LIN {X 0,Y 573.221,Z 379.814,A -85,B 0,C 180,E1 -2075.627,E2 -2075.627} C_VEL
LIN {X 0,Y 573.157,Z 385.848,A -85,B 0,C 180,E1 -2078.46,E2 -2078.46} C_VEL
LIN {X 0,Y 573.104,Z 392.081,A -85,B 0,C 180,E1 -2081.313,E2 -2081.313} C_VEL
LIN {X 0,Y 573.094,Z 398.89,A -85,B 0,C 180,E1 -2084.352,E2 -2084.352} C_VEL
LIN {X 0,Y 573.007,Z 405.201,A -85,B 0,C 180,E1 -2087.117,E2 -2087.117} C_VEL
LIN {X 0,Y 572.989,Z 410.326,A -85,B 0,C 180,E1 -2089.338,E2 -2089.338} C_VEL
LIN {X 0,Y 572.956,Z 415.575,A -85,B 0,C 180,E1 -2091.589,E2 -2091.589} C_VEL
LIN {X 0,Y 572.996,Z 419.359,A -85,B 0,C 180,E1 -2093.203,E2 -2093.203} C_VEL
LIN {X 0,Y 573.514,Z 425.872,A -85,B 0,C 180,E1 -2093.384,E2 -2093.384} C_VEL
LIN {X 0,Y 573.391,Z 435.633,A -85,B 0,C 180,E1 -2093.712,E2 -2093.712} C_VEL
LIN {X 0,Y 573.301,Z 447.019,A -85,B 0,C 180,E1 -2094.245,E2 -2094.245} C_VEL
LIN {X 0,Y 573.212,Z 457.823,A -85,B 0,C 180,E1 -2094.94,E2 -2094.94} C_VEL
LIN {X 0,Y 573.204,Z 465.961,A -85,B 0,C 180,E1 -2095.605,E2 -2095.605} C_VEL
LIN {X 0,Y 573.121,Z 474.398,A -85,B 0,C 180,E1 -2096.47,E2 -2096.47} C_VEL
LIN {X 0,Y 573.107,Z 481.387,A -85,B 0,C 180,E1 -2097.376,E2 -2097.376} C_VEL
LIN {X 0,Y 573.042,Z 486.731,A -85,B 0,C 180,E1 -2098.251,E2 -2098.251} C_VEL
LIN {X 0,Y 572.997,Z 492.29,A -85,B 0,C 180,E1 -2099.444,E2 -2099.444} C_VEL
LIN {X 0,Y 572.972,Z 494.817,A -85,B 0,C 180,E1 -2100.189,E2 -2100.189} C_VEL
LIN {X 0,Y 572.968,Z 496.858,A -85,B 0,C 180,E1 -2101.006,E2 -2101.006} C_VEL
LIN {X 0,Y 572.948,Z 498.62,A -85,B 0,C 180,E1 -2102.18,E2 -2102.18} C_VEL
LIN {X 0,Y 572.953,Z 498.823,A -85,B 0,C 180,E1 -2103.5,E2 -2103.5} C_VEL
LIN {X 0,Y 572.955,Z 497.535,A -85,B 0,C 180,E1 -2104.731,E2 -2104.731} C_VEL
LIN {X 0,Y 572.995,Z 494.283,A -85,B 0,C 180,E1 -2106.065,E2 -2106.065} C_VEL
LIN {X 0,Y 573.008,Z 490.226,A -85,B 0,C 180,E1 -2107.134,E2 -2107.134} C_VEL
LIN {X 0,Y 573.067,Z 484.148,A -85,B 0,C 180,E1 -2108.29,E2 -2108.29} C_VEL
LIN {X 0,Y 573.107,Z 477.566,A -85,B 0,C 180,E1 -2109.237,E2 -2109.237} C_VEL
LIN {X 0,Y 573.156,Z 469.185,A -85,B 0,C 180,E1 -2110.182,E2 -2110.182} C_VEL
LIN {X 0,Y 573.23,Z 459.968,A -85,B 0,C 180,E1 -2110.987,E2 -2110.987} C_VEL
LIN {X 0,Y 573.289,Z 451.126,A -85,B 0,C 180,E1 -2111.6,E2 -2111.6} C_VEL
LIN {X 0,Y 573.399,Z 441.637,A -85,B 0,C 180,E1 -2112.115,E2 -2112.115} C_VEL
LIN {X 0,Y 573.462,Z 430.782,A -85,B 0,C 180,E1 -2112.559,E2 -2112.559} C_VEL
LIN {X 0,Y 573.262,Z 421.712,A -85,B 0,C 180,E1 -2112.823,E2 -2112.823} C_VEL
LIN {X 0,Y 572.984,Z 419.34,A -85,B 0,C 180,E1 -2112.895,E2 -2112.895} C_VEL
LIN {X 0,Y 573.006,Z 412.902,A -85,B 0,C 180,E1 -2115.644,E2 -2115.644} C_VEL
LIN {X 0,Y 572.99,Z 406.238,A -85,B 0,C 180,E1 -2118.522,E2 -2118.522} C_VEL
LIN {X 0,Y 573.032,Z 398.959,A -85,B 0,C 180,E1 -2121.71,E2 -2121.71} C_VEL
LIN {X 0,Y 573.049,Z 393.732,A -85,B 0,C 180,E1 -2124.037,E2 -2124.037} C_VEL
LIN {X 0,Y 573.082,Z 388.318,A -85,B 0,C 180,E1 -2126.506,E2 -2126.506} C_VEL
LIN {X 0,Y 573.121,Z 382.746,A -85,B 0,C 180,E1 -2129.131,E2 -2129.131} C_VEL
LIN {X 0,Y 573.217,Z 376.758,A -85,B 0,C 180,E1 -2131.972,E2 -2131.972} C_VEL
LIN {X 0,Y 573.242,Z 371.144,A -85,B 0,C 180,E1 -2134.59,E2 -2134.59} C_VEL
LIN {X 0,Y 573.271,Z 369.078,A -85,B 0,C 180,E1 -2135.656,E2 -2135.656} C_VEL
LIN {X 0,Y 573.247,Z 369.082,A -85,B 0,C 180,E1 -2137.663,E2 -2137.663} C_VEL
LIN {X 0,Y 573.255,Z 369.082,A -85,B 0,C 180,E1 -2140.727,E2 -2140.727} C_VEL
LIN {X 0,Y 573.237,Z 369.082,A -85,B 0,C 180,E1 -2143.622,E2 -2143.622} C_VEL
LIN {X 0,Y 573.268,Z 369.08,A -85,B 0,C 180,E1 -2145.807,E2 -2145.807} C_VEL
LIN {X 0,Y 573.31,Z 369.075,A -85,B 0,C 180,E1 -2148.707,E2 -2148.707} C_VEL
LIN {X 0,Y 573.286,Z 369.076,A -85,B 0,C 180,E1 -2151.541,E2 -2151.541} C_VEL
LIN {X 0,Y 573.287,Z 369.075,A -85,B 0,C 180,E1 -2154.372,E2 -2154.372} C_VEL
LIN {X 0,Y 573.302,Z 369.076,A -85,B 0,C 180,E1 -2157.893,E2 -2157.893} C_VEL
LIN {X 0,Y 573.324,Z 369.073,A -85,B 0,C 180,E1 -2160.703,E2 -2160.703} C_VEL
LIN {X 0,Y 573.23,Z 369.083,A -85,B 0,C 180,E1 -2163.515,E2 -2163.515} C_VEL
LIN {X 0,Y 573.289,Z 369.075,A -85,B 0,C 180,E1 -2165.628,E2 -2165.628} C_VEL
LIN {X 0,Y 573.287,Z 369.076,A -85,B 0,C 180,E1 -2168.46,E2 -2168.46} C_VEL
LIN {X 0,Y 573.301,Z 369.077,A -85,B 0,C 180,E1 -2171.312,E2 -2171.312} C_VEL
LIN {X 0,Y 573.273,Z 369.076,A -85,B 0,C 180,E1 -2174.432,E2 -2174.432} C_VEL
LIN {X 0,Y 573.279,Z 369.075,A -85,B 0,C 180,E1 -2177.111,E2 -2177.111} C_VEL
LIN {X 0,Y 573.24,Z 369.08,A -85,B 0,C 180,E1 -2180.077,E2 -2180.077} C_VEL
LIN {X 0,Y 573.249,Z 369.081,A -85,B 0,C 180,E1 -2183.155,E2 -2183.155} C_VEL
LIN {X 0,Y 573.27,Z 369.078,A -85,B 0,C 180,E1 -2186.19,E2 -2186.19} C_VEL
LIN {X 0,Y 573.223,Z 369.085,A -85,B 0,C 180,E1 -2188.566,E2 -2188.566} C_VEL
LIN {X 0,Y 573.225,Z 369.082,A -85,B 0,C 180,E1 -2190.994,E2 -2190.994} C_VEL
LIN {X 0,Y 573.269,Z 369.076,A -85,B 0,C 180,E1 -2193.53,E2 -2193.53} C_VEL
LIN {X 0,Y 573.243,Z 369.079,A -85,B 0,C 180,E1 -2196.05,E2 -2196.05} C_VEL
LIN {X 0,Y 573.236,Z 369.08,A -85,B 0,C 180,E1 -2198.702,E2 -2198.702} C_VEL
LIN {X 0,Y 573.238,Z 369.081,A -85,B 0,C 180,E1 -2201.598,E2 -2201.598} C_VEL
LIN {X 0,Y 573.224,Z 369.083,A -85,B 0,C 180,E1 -2204.335,E2 -2204.335} C_VEL
LIN {X 0,Y 573.231,Z 369.085,A -85,B 0,C 180,E1 -2207.36,E2 -2207.36} C_VEL
LIN {X 0,Y 573.237,Z 369.082,A -85,B 0,C 180,E1 -2210.395,E2 -2210.395} C_VEL
LIN {X 0,Y 573.246,Z 369.081,A -85,B 0,C 180,E1 -2213.08,E2 -2213.08} C_VEL
LIN {X 0,Y 573.267,Z 369.079,A -85,B 0,C 180,E1 -2215.674,E2 -2215.674} C_VEL
LIN {X 0,Y 573.24,Z 369.084,A -85,B 0,C 180,E1 -2218.187,E2 -2218.187} C_VEL
LIN {X 0,Y 573.243,Z 369.126,A -85,B 0,C 180,E1 -2219.116,E2 -2219.116} C_VEL
LIN {X 0,Y 573.904,Z 373.266,A -85,B 0,C 180,E1 -2220.177,E2 -2220.177} C_VEL
LIN {X 0,Y 573.767,Z 383.575,A -85,B 0,C 180,E1 -2222.658,E2 -2222.658} C_VEL
LIN {X 0,Y 573.64,Z 393.801,A -85,B 0,C 180,E1 -2225.043,E2 -2225.043} C_VEL
LIN {X 0,Y 573.492,Z 407.081,A -85,B 0,C 180,E1 -2228.054,E2 -2228.054} C_VEL
LIN {X 0,Y 573.386,Z 420.619,A -85,B 0,C 180,E1 -2231.066,E2 -2231.066} C_VEL
LIN {X 0,Y 573.26,Z 433.998,A -85,B 0,C 180,E1 -2233.99,E2 -2233.99} C_VEL
LIN {X 0,Y 573.184,Z 445.774,A -85,B 0,C 180,E1 -2236.53,E2 -2236.53} C_VEL
LIN {X 0,Y 573.138,Z 450.085,A -85,B 0,C 180,E1 -2237.453,E2 -2237.453} C_VEL
LIN {X 0,Y 573.866,Z 456.184,A -85,B 0,C 180,E1 -2237.581,E2 -2237.581} C_VEL
LIN {X 0,Y 573.81,Z 469.797,A -85,B 0,C 180,E1 -2237.917,E2 -2237.917} C_VEL
LIN {X 0,Y 573.663,Z 481.536,A -85,B 0,C 180,E1 -2238.34,E2 -2238.34} C_VEL
LIN {X 0,Y 573.553,Z 492.943,A -85,B 0,C 180,E1 -2238.89,E2 -2238.89} C_VEL
LIN {X 0,Y 573.427,Z 504.229,A -85,B 0,C 180,E1 -2239.587,E2 -2239.587} C_VEL
LIN {X 0,Y 573.333,Z 514.621,A -85,B 0,C 180,E1 -2240.387,E2 -2240.387} C_VEL
LIN {X 0,Y 573.24,Z 523.131,A -85,B 0,C 180,E1 -2241.186,E2 -2241.186} C_VEL
LIN {X 0,Y 573.159,Z 530.975,A -85,B 0,C 180,E1 -2242.073,E2 -2242.073} C_VEL
LIN {X 0,Y 573.068,Z 538.985,A -85,B 0,C 180,E1 -2243.19,E2 -2243.19} C_VEL
LIN {X 0,Y 573.07,Z 545.688,A -85,B 0,C 180,E1 -2244.371,E2 -2244.371} C_VEL
LIN {X 0,Y 573.028,Z 550.378,A -85,B 0,C 180,E1 -2245.429,E2 -2245.429} C_VEL
LIN {X 0,Y 573.022,Z 553.963,A -85,B 0,C 180,E1 -2246.486,E2 -2246.486} C_VEL
LIN {X 0,Y 572.959,Z 555.814,A -85,B 0,C 180,E1 -2247.189,E2 -2247.189} C_VEL
LIN {X 0,Y 572.939,Z 557.203,A -85,B 0,C 180,E1 -2247.893,E2 -2247.893} C_VEL
LIN {X 0,Y 572.94,Z 558.786,A -85,B 0,C 180,E1 -2249.299,E2 -2249.299} C_VEL
LIN {X 0,Y 572.938,Z 559,A -85,B 0,C 180,E1 -2250.002,E2 -2250.002} C_VEL
LIN {X 0,Y 572.946,Z 558.184,A -85,B 0,C 180,E1 -2251.407,E2 -2251.407} C_VEL
LIN {X 0,Y 572.94,Z 557.196,A -85,B 0,C 180,E1 -2252.11,E2 -2252.11} C_VEL
LIN {X 0,Y 572.959,Z 555.805,A -85,B 0,C 180,E1 -2252.814,E2 -2252.814} C_VEL
LIN {X 0,Y 573.015,Z 552.891,A -85,B 0,C 180,E1 -2253.869,E2 -2253.869} C_VEL
LIN {X 0,Y 572.963,Z 548.944,A -85,B 0,C 180,E1 -2254.927,E2 -2254.927} C_VEL
LIN {X 0,Y 573.065,Z 542.869,A -85,B 0,C 180,E1 -2256.162,E2 -2256.162} C_VEL
LIN {X 0,Y 573.121,Z 536.228,A -85,B 0,C 180,E1 -2257.222,E2 -2257.222} C_VEL
LIN {X 0,Y 573.2,Z 527.979,A -85,B 0,C 180,E1 -2258.285,E2 -2258.285} C_VEL
LIN {X 0,Y 573.288,Z 519.524,A -85,B 0,C 180,E1 -2259.172,E2 -2259.172} C_VEL
LIN {X 0,Y 573.418,Z 509.08,A -85,B 0,C 180,E1 -2260.06,E2 -2260.06} C_VEL
LIN {X 0,Y 573.518,Z 497.505,A -85,B 0,C 180,E1 -2260.849,E2 -2260.849} C_VEL
LIN {X 0,Y 573.614,Z 485.855,A -85,B 0,C 180,E1 -2261.467,E2 -2261.467} C_VEL
LIN {X 0,Y 573.742,Z 473.141,A -85,B 0,C 180,E1 -2261.976,E2 -2261.976} C_VEL
LIN {X 0,Y 573.846,Z 460.469,A -85,B 0,C 180,E1 -2262.332,E2 -2262.332} C_VEL
LIN {X 0,Y 573.702,Z 453.526,A -85,B 0,C 180,E1 -2262.47,E2 -2262.47} C_VEL
LIN {X 0,Y 573.141,Z 450.07,A -85,B 0,C 180,E1 -2262.55,E2 -2262.55} C_VEL
LIN {X 0,Y 573.219,Z 437.347,A -85,B 0,C 180,E1 -2265.285,E2 -2265.285} C_VEL
LIN {X 0,Y 573.317,Z 425.571,A -85,B 0,C 180,E1 -2267.847,E2 -2267.847} C_VEL
LIN {X 0,Y 573.428,Z 413.795,A -85,B 0,C 180,E1 -2270.446,E2 -2270.446} C_VEL
LIN {X 0,Y 573.538,Z 401.461,A -85,B 0,C 180,E1 -2273.214,E2 -2273.214} C_VEL
LIN {X 0,Y 573.677,Z 390.192,A -85,B 0,C 180,E1 -2275.78,E2 -2275.78} C_VEL
LIN {X 0,Y 573.807,Z 378.43,A -85,B 0,C 180,E1 -2278.535,E2 -2278.535} C_VEL
LIN {X 0,Y 573.776,Z 371.893,A -85,B 0,C 180,E1 -2280.146,E2 -2280.146} C_VEL
LIN {X 0,Y 573.242,Z 369.084,A -85,B 0,C 180,E1 -2280.937,E2 -2280.937} C_VEL
LIN {X 0,Y 573.27,Z 369.074,A -85,B 0,C 180,E1 -2283.524,E2 -2283.524} C_VEL
LIN {X 0,Y 573.2,Z 369.085,A -85,B 0,C 180,E1 -2286.053,E2 -2286.053} C_VEL
LIN {X 0,Y 573.241,Z 369.078,A -85,B 0,C 180,E1 -2288.703,E2 -2288.703} C_VEL
LIN {X 0,Y 573.206,Z 369.084,A -85,B 0,C 180,E1 -2291.46,E2 -2291.46} C_VEL
LIN {X 0,Y 573.208,Z 369.08,A -85,B 0,C 180,E1 -2294.337,E2 -2294.337} C_VEL
LIN {X 0,Y 573.225,Z 369.083,A -85,B 0,C 180,E1 -2297.361,E2 -2297.361} C_VEL
LIN {X 0,Y 573.241,Z 369.079,A -85,B 0,C 180,E1 -2300.392,E2 -2300.392} C_VEL
LIN {X 0,Y 573.257,Z 369.075,A -85,B 0,C 180,E1 -2303.078,E2 -2303.078} C_VEL
LIN {X 0,Y 573.266,Z 369.075,A -85,B 0,C 180,E1 -2305.671,E2 -2305.671} C_VEL
LIN {X 0,Y 573.241,Z 369.08,A -85,B 0,C 180,E1 -2308.184,E2 -2308.184} C_VEL
LIN {X 0,Y 573.242,Z 369.076,A -85,B 0,C 180,E1 -2310.633,E2 -2310.633} C_VEL
LIN {X 0,Y 573.193,Z 369.087,A -85,B 0,C 180,E1 -2313.517,E2 -2313.517} C_VEL
LIN {X 0,Y 573.198,Z 369.081,A -85,B 0,C 180,E1 -2316.133,E2 -2316.133} C_VEL
LIN {X 0,Y 573.255,Z 369.082,A -85,B 0,C 180,E1 -2318.709,E2 -2318.709} C_VEL
LIN {X 0,Y 573.223,Z 369.078,A -85,B 0,C 180,E1 -2321.411,E2 -2321.411} C_VEL
LIN {X 0,Y 573.251,Z 369.077,A -85,B 0,C 180,E1 -2323.621,E2 -2323.621} C_VEL
LIN {X 0,Y 573.274,Z 369.08,A -85,B 0,C 180,E1 -2325.807,E2 -2325.807} C_VEL
LIN {X 0,Y 573.266,Z 369.074,A -85,B 0,C 180,E1 -2328.745,E2 -2328.745} C_VEL
LIN {X 0,Y 573.231,Z 369.081,A -85,B 0,C 180,E1 -2331.539,E2 -2331.539} C_VEL
LIN {X 0,Y 573.272,Z 369.075,A -85,B 0,C 180,E1 -2334.371,E2 -2334.371} C_VEL
LIN {X 0,Y 573.12,Z 369.184,A -85,B 0,C 180,E1 -2336.792,E2 -2336.792} C_VEL
LIN {X 0,Y 573.176,Z 375.949,A -85,B 0,C 180,E1 -2339.297,E2 -2339.297} C_VEL
LIN {X 0,Y 573.181,Z 381.47,A -85,B 0,C 180,E1 -2341.405,E2 -2341.405} C_VEL
LIN {X 0,Y 573.181,Z 388.472,A -85,B 0,C 180,E1 -2344.219,E2 -2344.219} C_VEL
LIN {X 0,Y 573.166,Z 394.594,A -85,B 0,C 180,E1 -2346.685,E2 -2346.685} C_VEL
LIN {X 0,Y 573.132,Z 400.488,A -85,B 0,C 180,E1 -2349.173,E2 -2349.173} C_VEL
LIN {X 0,Y 573.085,Z 407.375,A -85,B 0,C 180,E1 -2352.033,E2 -2352.033} C_VEL
LIN {X 0,Y 573.044,Z 414.457,A -85,B 0,C 180,E1 -2354.925,E2 -2354.925} C_VEL
LIN {X 0,Y 572.995,Z 419.903,A -85,B 0,C 180,E1 -2357.119,E2 -2357.119} C_VEL
LIN {X 0,Y 572.996,Z 423.478,A -85,B 0,C 180,E1 -2358.55,E2 -2358.55} C_VEL
LIN {X 0,Y 573.845,Z 430.186,A -85,B 0,C 180,E1 -2358.706,E2 -2358.706} C_VEL
LIN {X 0,Y 573.763,Z 442.032,A -85,B 0,C 180,E1 -2359.034,E2 -2359.034} C_VEL
LIN {X 0,Y 573.627,Z 453.34,A -85,B 0,C 180,E1 -2359.468,E2 -2359.468} C_VEL
LIN {X 0,Y 573.555,Z 463.451,A -85,B 0,C 180,E1 -2359.963,E2 -2359.963} C_VEL
LIN {X 0,Y 573.438,Z 474.178,A -85,B 0,C 180,E1 -2360.631,E2 -2360.631} C_VEL
LIN {X 0,Y 573.412,Z 475.368,A -85,B 0,C 180,E1 -2360.713,E2 -2360.713} C_VEL
LIN {X 0,Y 572.656,Z 480.164,A -85,B 0,C 180,E1 -2361.052,E2 -2361.052} C_VEL
LIN {X 0,Y 569.689,Z 487.629,A -85,B 0,C 180,E1 -2361.64,E2 -2361.64} C_VEL
LIN {X 0,Y 566.796,Z 494.631,A -85,B 0,C 180,E1 -2362.291,E2 -2362.291} C_VEL
LIN {X 0,Y 566.15,Z 498.531,A -85,B 0,C 180,E1 -2362.727,E2 -2362.727} C_VEL
LIN {X 0,Y 566.032,Z 506.689,A -85,B 0,C 180,E1 -2363.799,E2 -2363.799} C_VEL
LIN {X 0,Y 565.963,Z 513.78,A -85,B 0,C 180,E1 -2364.974,E2 -2364.974} C_VEL
LIN {X 0,Y 565.925,Z 519.365,A -85,B 0,C 180,E1 -2366.159,E2 -2366.159} C_VEL
LIN {X 0,Y 565.911,Z 523.539,A -85,B 0,C 180,E1 -2367.355,E2 -2367.355} C_VEL
LIN {X 0,Y 565.879,Z 525.689,A -85,B 0,C 180,E1 -2368.16,E2 -2368.16} C_VEL
LIN {X 0,Y 565.852,Z 527.302,A -85,B 0,C 180,E1 -2368.972,E2 -2368.972} C_VEL
LIN {X 0,Y 565.87,Z 528.361,A -85,B 0,C 180,E1 -2369.788,E2 -2369.788} C_VEL
LIN {X 0,Y 565.867,Z 528.999,A -85,B 0,C 180,E1 -2371.021,E2 -2371.021} C_VEL
LIN {X 0,Y 565.848,Z 528.29,A -85,B 0,C 180,E1 -2372.372,E2 -2372.372} C_VEL
LIN {X 0,Y 565.875,Z 526.246,A -85,B 0,C 180,E1 -2373.682,E2 -2373.682} C_VEL
LIN {X 0,Y 565.884,Z 522.947,A -85,B 0,C 180,E1 -2374.946,E2 -2374.946} C_VEL
LIN {X 0,Y 565.94,Z 518.319,A -85,B 0,C 180,E1 -2376.177,E2 -2376.177} C_VEL
LIN {X 0,Y 566.013,Z 511.801,A -85,B 0,C 180,E1 -2377.475,E2 -2377.475} C_VEL
LIN {X 0,Y 566.031,Z 505.02,A -85,B 0,C 180,E1 -2378.534,E2 -2378.534} C_VEL
LIN {X 0,Y 566.13,Z 497.583,A -85,B 0,C 180,E1 -2379.48,E2 -2379.48} C_VEL
LIN {X 0,Y 566.268,Z 488.609,A -85,B 0,C 180,E1 -2380.416,E2 -2380.416} C_VEL
LIN {X 0,Y 566.369,Z 478.973,A -85,B 0,C 180,E1 -2381.24,E2 -2381.24} C_VEL
LIN {X 0,Y 566.461,Z 468.39,A -85,B 0,C 180,E1 -2381.976,E2 -2381.976} C_VEL
LIN {X 0,Y 566.598,Z 457.183,A -85,B 0,C 180,E1 -2382.593,E2 -2382.593} C_VEL
LIN {X 0,Y 566.786,Z 444.591,A -85,B 0,C 180,E1 -2383.12,E2 -2383.12} C_VEL
LIN {X 0,Y 566.924,Z 432.071,A -85,B 0,C 180,E1 -2383.492,E2 -2383.492} C_VEL
LIN {X 0,Y 566.55,Z 427.486,A -85,B 0,C 180,E1 -2383.602,E2 -2383.602} C_VEL
LIN {X 0,Y 565.911,Z 423.488,A -85,B 0,C 180,E1 -2383.695,E2 -2383.695} C_VEL
LIN {X 0,Y 565.921,Z 416.591,A -85,B 0,C 180,E1 -2386.499,E2 -2386.499} C_VEL
LIN {X 0,Y 565.949,Z 409.925,A -85,B 0,C 180,E1 -2389.244,E2 -2389.244} C_VEL
LIN {X 0,Y 565.991,Z 403.165,A -85,B 0,C 180,E1 -2392.073,E2 -2392.073} C_VEL
LIN {X 0,Y 566.075,Z 395.831,A -85,B 0,C 180,E1 -2395.172,E2 -2395.172} C_VEL
LIN {X 0,Y 566.094,Z 388.666,A -85,B 0,C 180,E1 -2398.153,E2 -2398.153} C_VEL
LIN {X 0,Y 566.089,Z 381.695,A -85,B 0,C 180,E1 -2401.04,E2 -2401.04} C_VEL
LIN {X 0,Y 566.091,Z 375.921,A -85,B 0,C 180,E1 -2403.452,E2 -2403.452} C_VEL
LIN {X 0,Y 566.204,Z 369.96,A -85,B 0,C 180,E1 -2405.916,E2 -2405.916} C_VEL
LIN {X 0,Y 566.21,Z 369.96,A -85,B 0,C 180,E1 -2408.901,E2 -2408.901} C_VEL
LIN {X 0,Y 566.189,Z 369.956,A -85,B 0,C 180,E1 -2411.171,E2 -2411.171} C_VEL
LIN {X 0,Y 566.212,Z 369.957,A -85,B 0,C 180,E1 -2413.411,E2 -2413.411} C_VEL
LIN {X 0,Y 566.198,Z 369.957,A -85,B 0,C 180,E1 -2416.358,E2 -2416.358} C_VEL
LIN {X 0,Y 566.236,Z 369.952,A -85,B 0,C 180,E1 -2418.674,E2 -2418.674} C_VEL
LIN {X 0,Y 566.227,Z 369.958,A -85,B 0,C 180,E1 -2421.433,E2 -2421.433} C_VEL
LIN {X 0,Y 566.254,Z 369.952,A -85,B 0,C 180,E1 -2424.3,E2 -2424.3} C_VEL
LIN {X 0,Y 566.28,Z 369.95,A -85,B 0,C 180,E1 -2427.865,E2 -2427.865} C_VEL
LIN {X 0,Y 566.295,Z 370.044,A -85,B 0,C 180,E1 -2430.532,E2 -2430.532} C_VEL
LIN {X 0,Y 566.195,Z 374.816,A -85,B 0,C 180,E1 -2432.844,E2 -2432.844} C_VEL
LIN {X 0,Y 566.172,Z 380.804,A -85,B 0,C 180,E1 -2435.697,E2 -2435.697} C_VEL
LIN {X 0,Y 566.083,Z 386.804,A -85,B 0,C 180,E1 -2438.566,E2 -2438.566} C_VEL
LIN {X 0,Y 566.035,Z 393.035,A -85,B 0,C 180,E1 -2441.457,E2 -2441.457} C_VEL
LIN {X 0,Y 566.019,Z 399.589,A -85,B 0,C 180,E1 -2444.422,E2 -2444.422} C_VEL
LIN {X 0,Y 565.924,Z 406.166,A -85,B 0,C 180,E1 -2447.338,E2 -2447.338} C_VEL
LIN {X 0,Y 565.91,Z 411.304,A -85,B 0,C 180,E1 -2449.589,E2 -2449.589} C_VEL
LIN {X 0,Y 565.873,Z 416.567,A -85,B 0,C 180,E1 -2451.873,E2 -2451.873} C_VEL
LIN {X 0,Y 565.912,Z 419.522,A -85,B 0,C 180,E1 -2453.087,E2 -2453.087} C_VEL
LIN {X 0,Y 566.523,Z 426.242,A -85,B 0,C 180,E1 -2453.274,E2 -2453.274} C_VEL
LIN {X 0,Y 566.391,Z 436.625,A -85,B 0,C 180,E1 -2453.635,E2 -2453.635} C_VEL
LIN {X 0,Y 566.268,Z 447.72,A -85,B 0,C 180,E1 -2454.175,E2 -2454.175} C_VEL
LIN {X 0,Y 566.176,Z 458.161,A -85,B 0,C 180,E1 -2454.863,E2 -2454.863} C_VEL
LIN {X 0,Y 566.15,Z 466.175,A -85,B 0,C 180,E1 -2455.533,E2 -2455.533} C_VEL
LIN {X 0,Y 566.05,Z 474.052,A -85,B 0,C 180,E1 -2456.348,E2 -2456.348} C_VEL
LIN {X 0,Y 566.01,Z 480.308,A -85,B 0,C 180,E1 -2457.15,E2 -2457.15} C_VEL
LIN {X 0,Y 565.949,Z 486.546,A -85,B 0,C 180,E1 -2458.154,E2 -2458.154} C_VEL
LIN {X 0,Y 565.924,Z 491.874,A -85,B 0,C 180,E1 -2459.291,E2 -2459.291} C_VEL
LIN {X 0,Y 565.891,Z 494.952,A -85,B 0,C 180,E1 -2460.195,E2 -2460.195} C_VEL
LIN {X 0,Y 565.839,Z 497.681,A -85,B 0,C 180,E1 -2461.441,E2 -2461.441} C_VEL
LIN {X 0,Y 565.841,Z 498.72,A -85,B 0,C 180,E1 -2462.372,E2 -2462.372} C_VEL
LIN {X 0,Y 565.836,Z 498.988,A -85,B 0,C 180,E1 -2463.125,E2 -2463.125} C_VEL
LIN {X 0,Y 565.855,Z 498.574,A -85,B 0,C 180,E1 -2463.977,E2 -2463.977} C_VEL
LIN {X 0,Y 565.847,Z 497.228,A -85,B 0,C 180,E1 -2464.942,E2 -2464.942} C_VEL
LIN {X 0,Y 565.917,Z 494.055,A -85,B 0,C 180,E1 -2466.175,E2 -2466.175} C_VEL
LIN {X 0,Y 565.927,Z 489.398,A -85,B 0,C 180,E1 -2467.365,E2 -2467.365} C_VEL
LIN {X 0,Y 565.984,Z 484.024,A -85,B 0,C 180,E1 -2468.376,E2 -2468.376} C_VEL
LIN {X 0,Y 566.024,Z 477.803,A -85,B 0,C 180,E1 -2469.286,E2 -2469.286} C_VEL
LIN {X 0,Y 566.099,Z 469.835,A -85,B 0,C 180,E1 -2470.205,E2 -2470.205} C_VEL
LIN {X 0,Y 566.169,Z 460.783,A -85,B 0,C 180,E1 -2471.022,E2 -2471.022} C_VEL
LIN {X 0,Y 566.269,Z 451.675,A -85,B 0,C 180,E1 -2471.671,E2 -2471.671} C_VEL
LIN {X 0,Y 566.366,Z 442.425,A -85,B 0,C 180,E1 -2472.19,E2 -2472.19} C_VEL
LIN {X 0,Y 566.459,Z 432.79,A -85,B 0,C 180,E1 -2472.603,E2 -2472.603} C_VEL
LIN {X 0,Y 566.371,Z 423.198,A -85,B 0,C 180,E1 -2472.903,E2 -2472.903} C_VEL
LIN {X 0,Y 565.917,Z 419.341,A -85,B 0,C 180,E1 -2473.019,E2 -2473.019} C_VEL
LIN {X 0,Y 565.917,Z 412.282,A -85,B 0,C 180,E1 -2476.075,E2 -2476.075} C_VEL
LIN {X 0,Y 565.902,Z 405.975,A -85,B 0,C 180,E1 -2478.837,E2 -2478.837} C_VEL
LIN {X 0,Y 565.954,Z 399.704,A -85,B 0,C 180,E1 -2481.619,E2 -2481.619} C_VEL
LIN {X 0,Y 565.962,Z 393.8,A -85,B 0,C 180,E1 -2484.294,E2 -2484.294} C_VEL
LIN {X 0,Y 566.031,Z 388.257,A -85,B 0,C 180,E1 -2486.886,E2 -2486.886} C_VEL
LIN {X 0,Y 566.061,Z 383.001,A -85,B 0,C 180,E1 -2489.4,E2 -2489.4} C_VEL
LIN {X 0,Y 566.162,Z 377.851,A -85,B 0,C 180,E1 -2491.855,E2 -2491.855} C_VEL
LIN {X 0,Y 566.204,Z 372.763,A -85,B 0,C 180,E1 -2494.251,E2 -2494.251} C_VEL
LIN {X 0,Y 566.219,Z 369.957,A -85,B 0,C 180,E1 -2495.625,E2 -2495.625} C_VEL
LIN {X 0,Y 566.192,Z 369.958,A -85,B 0,C 180,E1 -2498.576,E2 -2498.576} C_VEL
LIN {X 0,Y 566.198,Z 369.958,A -85,B 0,C 180,E1 -2501.172,E2 -2501.172} C_VEL
LIN {X 0,Y 566.189,Z 369.959,A -85,B 0,C 180,E1 -2504.153,E2 -2504.153} C_VEL
LIN {X 0,Y 566.19,Z 369.959,A -85,B 0,C 180,E1 -2506.359,E2 -2506.359} C_VEL
LIN {X 0,Y 566.256,Z 369.95,A -85,B 0,C 180,E1 -2509.271,E2 -2509.271} C_VEL
LIN {X 0,Y 566.223,Z 369.954,A -85,B 0,C 180,E1 -2512.153,E2 -2512.153} C_VEL
LIN {X 0,Y 566.272,Z 369.95,A -85,B 0,C 180,E1 -2515.016,E2 -2515.016} C_VEL
LIN {X 0,Y 566.271,Z 369.951,A -85,B 0,C 180,E1 -2517.866,E2 -2517.866} C_VEL
LIN {X 0,Y 566.292,Z 369.948,A -85,B 0,C 180,E1 -2520.711,E2 -2520.711} C_VEL
LIN {X 0,Y 566.26,Z 369.95,A -85,B 0,C 180,E1 -2522.846,E2 -2522.846} C_VEL
LIN {X 0,Y 566.256,Z 369.951,A -85,B 0,C 180,E1 -2525.699,E2 -2525.699} C_VEL
LIN {X 0,Y 566.23,Z 369.957,A -85,B 0,C 180,E1 -2528.566,E2 -2528.566} C_VEL
LIN {X 0,Y 566.24,Z 369.954,A -85,B 0,C 180,E1 -2531.455,E2 -2531.455} C_VEL
LIN {X 0,Y 566.224,Z 369.954,A -85,B 0,C 180,E1 -2534.513,E2 -2534.513} C_VEL
LIN {X 0,Y 566.235,Z 369.952,A -85,B 0,C 180,E1 -2537.331,E2 -2537.331} C_VEL
LIN {X 0,Y 566.202,Z 369.958,A -85,B 0,C 180,E1 -2540.338,E2 -2540.338} C_VEL
LIN {X 0,Y 566.208,Z 369.959,A -85,B 0,C 180,E1 -2543.403,E2 -2543.403} C_VEL
LIN {X 0,Y 566.204,Z 369.958,A -85,B 0,C 180,E1 -2545.75,E2 -2545.75} C_VEL
LIN {X 0,Y 566.187,Z 369.958,A -85,B 0,C 180,E1 -2548.205,E2 -2548.205} C_VEL
LIN {X 0,Y 566.177,Z 369.959,A -85,B 0,C 180,E1 -2550.593,E2 -2550.593} C_VEL
LIN {X 0,Y 566.21,Z 369.956,A -85,B 0,C 180,E1 -2553.103,E2 -2553.103} C_VEL
LIN {X 0,Y 566.195,Z 369.959,A -85,B 0,C 180,E1 -2555.69,E2 -2555.69} C_VEL
LIN {X 0,Y 566.202,Z 369.957,A -85,B 0,C 180,E1 -2558.561,E2 -2558.561} C_VEL
LIN {X 0,Y 566.196,Z 369.958,A -85,B 0,C 180,E1 -2561.138,E2 -2561.138} C_VEL
LIN {X 0,Y 566.186,Z 369.959,A -85,B 0,C 180,E1 -2564.037,E2 -2564.037} C_VEL
LIN {X 0,Y 566.192,Z 369.959,A -85,B 0,C 180,E1 -2567.084,E2 -2567.084} C_VEL
LIN {X 0,Y 566.215,Z 369.957,A -85,B 0,C 180,E1 -2569.805,E2 -2569.805} C_VEL
LIN {X 0,Y 566.188,Z 369.961,A -85,B 0,C 180,E1 -2572.601,E2 -2572.601} C_VEL
LIN {X 0,Y 566.213,Z 369.958,A -85,B 0,C 180,E1 -2575.185,E2 -2575.185} C_VEL
LIN {X 0,Y 566.224,Z 369.957,A -85,B 0,C 180,E1 -2577.746,E2 -2577.746} C_VEL
LIN {X 0,Y 566.227,Z 370.122,A -85,B 0,C 180,E1 -2578.918,E2 -2578.918} C_VEL
LIN {X 0,Y 566.998,Z 374.99,A -85,B 0,C 180,E1 -2580.188,E2 -2580.188} C_VEL
LIN {X 0,Y 566.775,Z 386.505,A -85,B 0,C 180,E1 -2583.011,E2 -2583.011} C_VEL
LIN {X 0,Y 566.604,Z 396.827,A -85,B 0,C 180,E1 -2585.45,E2 -2585.45} C_VEL
LIN {X 0,Y 566.501,Z 408.763,A -85,B 0,C 180,E1 -2588.152,E2 -2588.152} C_VEL
LIN {X 0,Y 566.337,Z 422.222,A -85,B 0,C 180,E1 -2591.179,E2 -2591.179} C_VEL
LIN {X 0,Y 566.229,Z 433.998,A -85,B 0,C 180,E1 -2593.786,E2 -2593.786} C_VEL
LIN {X 0,Y 566.11,Z 447.456,A -85,B 0,C 180,E1 -2596.724,E2 -2596.724} C_VEL
LIN {X 0,Y 566.083,Z 450.085,A -85,B 0,C 180,E1 -2597.294,E2 -2597.294} C_VEL
LIN {X 0,Y 566.959,Z 457.324,A -85,B 0,C 180,E1 -2597.45,E2 -2597.45} C_VEL
LIN {X 0,Y 566.863,Z 470.556,A -85,B 0,C 180,E1 -2597.789,E2 -2597.789} C_VEL
LIN {X 0,Y 566.7,Z 482.561,A -85,B 0,C 180,E1 -2598.24,E2 -2598.24} C_VEL
LIN {X 0,Y 566.548,Z 494.976,A -85,B 0,C 180,E1 -2598.868,E2 -2598.868} C_VEL
LIN {X 0,Y 566.434,Z 505.509,A -85,B 0,C 180,E1 -2599.547,E2 -2599.547} C_VEL
LIN {X 0,Y 566.3,Z 515.667,A -85,B 0,C 180,E1 -2600.357,E2 -2600.357} C_VEL
LIN {X 0,Y 566.165,Z 524.803,A -85,B 0,C 180,E1 -2601.255,E2 -2601.255} C_VEL
LIN {X 0,Y 566.079,Z 533.703,A -85,B 0,C 180,E1 -2602.332,E2 -2602.332} C_VEL
LIN {X 0,Y 565.966,Z 540.966,A -85,B 0,C 180,E1 -2603.424,E2 -2603.424} C_VEL
LIN {X 0,Y 566.003,Z 545.688,A -85,B 0,C 180,E1 -2604.301,E2 -2604.301} C_VEL
LIN {X 0,Y 565.933,Z 550.378,A -85,B 0,C 180,E1 -2605.372,E2 -2605.372} C_VEL
LIN {X 0,Y 565.926,Z 553.964,A -85,B 0,C 180,E1 -2606.442,E2 -2606.442} C_VEL
LIN {X 0,Y 565.877,Z 555.814,A -85,B 0,C 180,E1 -2607.154,E2 -2607.154} C_VEL
LIN {X 0,Y 565.846,Z 558.188,A -85,B 0,C 180,E1 -2608.578,E2 -2608.578} C_VEL
LIN {X 0,Y 565.839,Z 559,A -85,B 0,C 180,E1 -2610.002,E2 -2610.002} C_VEL
LIN {X 0,Y 565.846,Z 558.184,A -85,B 0,C 180,E1 -2611.425,E2 -2611.425} C_VEL
LIN {X 0,Y 565.878,Z 555.805,A -85,B 0,C 180,E1 -2612.849,E2 -2612.849} C_VEL
LIN {X 0,Y 565.927,Z 552.891,A -85,B 0,C 180,E1 -2613.918,E2 -2613.918} C_VEL
LIN {X 0,Y 565.878,Z 548.944,A -85,B 0,C 180,E1 -2614.989,E2 -2614.989} C_VEL
LIN {X 0,Y 566.002,Z 543.859,A -85,B 0,C 180,E1 -2616.06,E2 -2616.06} C_VEL
LIN {X 0,Y 566.042,Z 537.458,A -85,B 0,C 180,E1 -2617.134,E2 -2617.134} C_VEL
LIN {X 0,Y 566.134,Z 529.467,A -85,B 0,C 180,E1 -2618.209,E2 -2618.209} C_VEL
LIN {X 0,Y 566.23,Z 521.322,A -85,B 0,C 180,E1 -2619.107,E2 -2619.107} C_VEL
LIN {X 0,Y 566.347,Z 511.385,A -85,B 0,C 180,E1 -2620.006,E2 -2620.006} C_VEL
LIN {X 0,Y 566.518,Z 500.299,A -85,B 0,C 180,E1 -2620.807,E2 -2620.807} C_VEL
LIN {X 0,Y 566.611,Z 487.922,A -85,B 0,C 180,E1 -2621.511,E2 -2621.511} C_VEL
LIN {X 0,Y 566.78,Z 475.736,A -85,B 0,C 180,E1 -2622.034,E2 -2622.034} C_VEL
LIN {X 0,Y 566.922,Z 462.3,A -85,B 0,C 180,E1 -2622.44,E2 -2622.44} C_VEL
LIN {X 0,Y 566.751,Z 454.17,A -85,B 0,C 180,E1 -2622.616,E2 -2622.616} C_VEL
LIN {X 0,Y 566.086,Z 450.07,A -85,B 0,C 180,E1 -2622.709,E2 -2622.709} C_VEL
LIN {X 0,Y 566.177,Z 437.347,A -85,B 0,C 180,E1 -2625.48,E2 -2625.48} C_VEL
LIN {X 0,Y 566.299,Z 425.571,A -85,B 0,C 180,E1 -2628.076,E2 -2628.076} C_VEL
LIN {X 0,Y 566.416,Z 413.795,A -85,B 0,C 180,E1 -2630.71,E2 -2630.71} C_VEL
LIN {X 0,Y 566.568,Z 402.011,A -85,B 0,C 180,E1 -2633.388,E2 -2633.388} C_VEL
LIN {X 0,Y 566.702,Z 390.097,A -85,B 0,C 180,E1 -2636.121,E2 -2636.121} C_VEL
LIN {X 0,Y 566.876,Z 379.903,A -85,B 0,C 180,E1 -2638.573,E2 -2638.573} C_VEL
LIN {X 0,Y 566.873,Z 373.612,A -85,B 0,C 180,E1 -2640.14,E2 -2640.14} C_VEL
LIN {X 0,Y 566.179,Z 369.964,A -85,B 0,C 180,E1 -2641.113,E2 -2641.113} C_VEL
LIN {X 0,Y 566.219,Z 369.953,A -85,B 0,C 180,E1 -2643.735,E2 -2643.735} C_VEL
LIN {X 0,Y 566.188,Z 369.961,A -85,B 0,C 180,E1 -2646.572,E2 -2646.572} C_VEL
LIN {X 0,Y 566.217,Z 369.955,A -85,B 0,C 180,E1 -2649.686,E2 -2649.686} C_VEL
LIN {X 0,Y 566.15,Z 369.96,A -85,B 0,C 180,E1 -2652.911,E2 -2652.911} C_VEL
LIN {X 0,Y 566.158,Z 369.958,A -85,B 0,C 180,E1 -2656.054,E2 -2656.054} C_VEL
LIN {X 0,Y 566.17,Z 369.964,A -85,B 0,C 180,E1 -2658.86,E2 -2658.86} C_VEL
LIN {X 0,Y 566.212,Z 369.951,A -85,B 0,C 180,E1 -2661.443,E2 -2661.443} C_VEL
LIN {X 0,Y 566.168,Z 369.965,A -85,B 0,C 180,E1 -2664.308,E2 -2664.308} C_VEL
LIN {X 0,Y 566.208,Z 369.952,A -85,B 0,C 180,E1 -2666.897,E2 -2666.897} C_VEL
LIN {X 0,Y 566.174,Z 369.96,A -85,B 0,C 180,E1 -2669.407,E2 -2669.407} C_VEL
LIN {X 0,Y 566.174,Z 369.96,A -85,B 0,C 180,E1 -2671.855,E2 -2671.855} C_VEL
LIN {X 0,Y 566.171,Z 369.957,A -85,B 0,C 180,E1 -2674.249,E2 -2674.249} C_VEL
LIN {X 0,Y 566.175,Z 369.958,A -85,B 0,C 180,E1 -2677.368,E2 -2677.368} C_VEL
LIN {X 0,Y 566.209,Z 369.952,A -85,B 0,C 180,E1 -2679.662,E2 -2679.662} C_VEL
LIN {X 0,Y 566.203,Z 369.956,A -85,B 0,C 180,E1 -2682.668,E2 -2682.668} C_VEL
LIN {X 0,Y 566.236,Z 369.954,A -85,B 0,C 180,E1 -2685.627,E2 -2685.627} C_VEL
LIN {X 0,Y 566.237,Z 369.949,A -85,B 0,C 180,E1 -2688.676,E2 -2688.676} C_VEL
LIN {X 0,Y 566.186,Z 369.96,A -85,B 0,C 180,E1 -2691.433,E2 -2691.433} C_VEL
LIN {X 0,Y 566.239,Z 369.951,A -85,B 0,C 180,E1 -2694.301,E2 -2694.301} C_VEL
LIN {X 0,Y 566.058,Z 370.033,A -85,B 0,C 180,E1 -2696.841,E2 -2696.841} C_VEL
LIN {X 0,Y 566.146,Z 378.45,A -85,B 0,C 180,E1 -2700,E2 -2700} C_VEL
LIN {X 0,Y 566.082,Z 385.71,A -85,B 0,C 180,E1 -2702.846,E2 -2702.846} C_VEL
LIN {X 0,Y 566.144,Z 391.062,A -85,B 0,C 180,E1 -2704.985,E2 -2704.985} C_VEL
LIN {X 0,Y 566.081,Z 398.004,A -85,B 0,C 180,E1 -2707.849,E2 -2707.849} C_VEL
LIN {X 0,Y 566.032,Z 404.861,A -85,B 0,C 180,E1 -2710.733,E2 -2710.733} C_VEL
LIN {X 0,Y 565.981,Z 411.856,A -85,B 0,C 180,E1 -2713.646,E2 -2713.646} C_VEL
LIN {X 0,Y 565.93,Z 419.052,A -85,B 0,C 180,E1 -2716.596,E2 -2716.596} C_VEL
LIN {X 0,Y 565.921,Z 423.479,A -85,B 0,C 180,E1 -2718.391,E2 -2718.391} C_VEL
LIN {X 0,Y 566.918,Z 430.796,A -85,B 0,C 180,E1 -2718.569,E2 -2718.569} C_VEL
LIN {X 0,Y 566.804,Z 442.349,A -85,B 0,C 180,E1 -2718.896,E2 -2718.896} C_VEL
LIN {X 0,Y 566.657,Z 453.794,A -85,B 0,C 180,E1 -2719.345,E2 -2719.345} C_VEL
LIN {X 0,Y 566.559,Z 463.924,A -85,B 0,C 180,E1 -2719.851,E2 -2719.851} C_VEL
LIN {X 0,Y 566.436,Z 474.413,A -85,B 0,C 180,E1 -2720.518,E2 -2720.518} C_VEL
LIN {X 0,Y 566.314,Z 485.153,A -85,B 0,C 180,E1 -2721.359,E2 -2721.359} C_VEL
LIN {X 0,Y 566.209,Z 494.303,A -85,B 0,C 180,E1 -2722.245,E2 -2722.245} C_VEL
LIN {X 0,Y 566.15,Z 498.531,A -85,B 0,C 180,E1 -2722.727,E2 -2722.727} C_VEL
LIN {X 0,Y 565.486,Z 502.32,A -85,B 0,C 180,E1 -2723.182,E2 -2723.182} C_VEL
LIN {X 0,Y 562.523,Z 508.004,A -85,B 0,C 180,E1 -2723.952,E2 -2723.952} C_VEL
LIN {X 0,Y 559.544,Z 513.102,A -85,B 0,C 180,E1 -2724.774,E2 -2724.774} C_VEL
LIN {X 0,Y 558.864,Z 515.801,A -85,B 0,C 180,E1 -2725.305,E2 -2725.305} C_VEL
LIN {X 0,Y 558.846,Z 520.67,A -85,B 0,C 180,E1 -2726.434,E2 -2726.434} C_VEL
LIN {X 0,Y 558.793,Z 524.77,A -85,B 0,C 180,E1 -2727.733,E2 -2727.733} C_VEL
LIN {X 0,Y 558.753,Z 526.584,A -85,B 0,C 180,E1 -2728.552,E2 -2728.552} C_VEL
LIN {X 0,Y 558.771,Z 528.379,A -85,B 0,C 180,E1 -2729.789,E2 -2729.789} C_VEL
LIN {X 0,Y 558.764,Z 528.971,A -85,B 0,C 180,E1 -2731.208,E2 -2731.208} C_VEL
LIN {X 0,Y 558.763,Z 528.091,A -85,B 0,C 180,E1 -2732.572,E2 -2732.572} C_VEL
LIN {X 0,Y 558.781,Z 525.895,A -85,B 0,C 180,E1 -2733.89,E2 -2733.89} C_VEL
LIN {X 0,Y 558.8,Z 522.39,A -85,B 0,C 180,E1 -2735.164,E2 -2735.164} C_VEL
LIN {X 0,Y 558.855,Z 517.611,A -85,B 0,C 180,E1 -2736.404,E2 -2736.404} C_VEL
LIN {X 0,Y 558.924,Z 511.504,A -85,B 0,C 180,E1 -2737.61,E2 -2737.61} C_VEL
LIN {X 0,Y 558.993,Z 503.895,A -85,B 0,C 180,E1 -2738.784,E2 -2738.784} C_VEL
LIN {X 0,Y 559.123,Z 495.09,A -85,B 0,C 180,E1 -2739.87,E2 -2739.87} C_VEL
LIN {X 0,Y 559.263,Z 485.735,A -85,B 0,C 180,E1 -2740.803,E2 -2740.803} C_VEL
LIN {X 0,Y 559.394,Z 475.179,A -85,B 0,C 180,E1 -2741.655,E2 -2741.655} C_VEL
LIN {X 0,Y 559.529,Z 463.549,A -85,B 0,C 180,E1 -2742.403,E2 -2742.403} C_VEL
LIN {X 0,Y 559.722,Z 451.047,A -85,B 0,C 180,E1 -2743.019,E2 -2743.019} C_VEL
LIN {X 0,Y 559.915,Z 438.18,A -85,B 0,C 180,E1 -2743.483,E2 -2743.483} C_VEL
LIN {X 0,Y 559.799,Z 429.29,A -85,B 0,C 180,E1 -2743.717,E2 -2743.717} C_VEL
LIN {X 0,Y 558.819,Z 423.473,A -85,B 0,C 180,E1 -2743.865,E2 -2743.865} C_VEL
LIN {X 0,Y 558.857,Z 416.264,A -85,B 0,C 180,E1 -2746.835,E2 -2746.835} C_VEL
LIN {X 0,Y 558.904,Z 409.551,A -85,B 0,C 180,E1 -2749.639,E2 -2749.639} C_VEL
LIN {X 0,Y 558.924,Z 403.053,A -85,B 0,C 180,E1 -2752.389,E2 -2752.389} C_VEL
LIN {X 0,Y 559.017,Z 397.361,A -85,B 0,C 180,E1 -2754.804,E2 -2754.804} C_VEL
LIN {X 0,Y 559.033,Z 391.266,A -85,B 0,C 180,E1 -2757.384,E2 -2757.384} C_VEL
LIN {X 0,Y 559.008,Z 385.443,A -85,B 0,C 180,E1 -2759.808,E2 -2759.808} C_VEL
LIN {X 0,Y 559.044,Z 379.588,A -85,B 0,C 180,E1 -2762.279,E2 -2762.279} C_VEL
LIN {X 0,Y 559.102,Z 371.833,A -85,B 0,C 180,E1 -2765.491,E2 -2765.491} C_VEL
LIN {X 0,Y 559.179,Z 370.834,A -85,B 0,C 180,E1 -2765.988,E2 -2765.988} C_VEL
LIN {X 0,Y 559.175,Z 370.833,A -85,B 0,C 180,E1 -2768.623,E2 -2768.623} C_VEL
LIN {X 0,Y 559.158,Z 370.833,A -85,B 0,C 180,E1 -2770.925,E2 -2770.925} C_VEL
LIN {X 0,Y 559.165,Z 370.833,A -85,B 0,C 180,E1 -2773.947,E2 -2773.947} C_VEL
LIN {X 0,Y 559.173,Z 370.831,A -85,B 0,C 180,E1 -2776.183,E2 -2776.183} C_VEL
LIN {X 0,Y 559.193,Z 370.828,A -85,B 0,C 180,E1 -2779.132,E2 -2779.132} C_VEL
LIN {X 0,Y 559.205,Z 370.827,A -85,B 0,C 180,E1 -2782.052,E2 -2782.052} C_VEL
LIN {X 0,Y 559.241,Z 370.824,A -85,B 0,C 180,E1 -2784.952,E2 -2784.952} C_VEL
LIN {X 0,Y 559.251,Z 370.826,A -85,B 0,C 180,E1 -2787.838,E2 -2787.838} C_VEL
LIN {X 0,Y 559.268,Z 370.991,A -85,B 0,C 180,E1 -2790.538,E2 -2790.538} C_VEL
LIN {X 0,Y 559.142,Z 375.793,A -85,B 0,C 180,E1 -2792.88,E2 -2792.88} C_VEL
LIN {X 0,Y 559.125,Z 381.785,A -85,B 0,C 180,E1 -2795.769,E2 -2795.769} C_VEL
LIN {X 0,Y 559.02,Z 387.855,A -85,B 0,C 180,E1 -2798.675,E2 -2798.675} C_VEL
LIN {X 0,Y 558.998,Z 393.395,A -85,B 0,C 180,E1 -2801.29,E2 -2801.29} C_VEL
LIN {X 0,Y 558.937,Z 400.44,A -85,B 0,C 180,E1 -2804.563,E2 -2804.563} C_VEL
LIN {X 0,Y 558.838,Z 407.133,A -85,B 0,C 180,E1 -2807.565,E2 -2807.565} C_VEL
LIN {X 0,Y 558.813,Z 412.285,A -85,B 0,C 180,E1 -2809.848,E2 -2809.848} C_VEL
LIN {X 0,Y 558.784,Z 417.563,A -85,B 0,C 180,E1 -2812.165,E2 -2812.165} C_VEL
LIN {X 0,Y 558.805,Z 419.591,A -85,B 0,C 180,E1 -2812.961,E2 -2812.961} C_VEL
LIN {X 0,Y 559.544,Z 426.381,A -85,B 0,C 180,E1 -2813.155,E2 -2813.155} C_VEL
LIN {X 0,Y 559.388,Z 435.886,A -85,B 0,C 180,E1 -2813.487,E2 -2813.487} C_VEL
LIN {X 0,Y 559.262,Z 446.702,A -85,B 0,C 180,E1 -2814.004,E2 -2814.004} C_VEL
LIN {X 0,Y 559.16,Z 457.321,A -85,B 0,C 180,E1 -2814.696,E2 -2814.696} C_VEL
LIN {X 0,Y 559.102,Z 465.762,A -85,B 0,C 180,E1 -2815.399,E2 -2815.399} C_VEL
LIN {X 0,Y 558.989,Z 472.676,A -85,B 0,C 180,E1 -2816.104,E2 -2816.104} C_VEL
LIN {X 0,Y 558.939,Z 479.147,A -85,B 0,C 180,E1 -2816.912,E2 -2816.912} C_VEL
LIN {X 0,Y 558.847,Z 484.484,A -85,B 0,C 180,E1 -2817.728,E2 -2817.728} C_VEL
LIN {X 0,Y 558.833,Z 488.83,A -85,B 0,C 180,E1 -2818.545,E2 -2818.545} C_VEL
LIN {X 0,Y 558.846,Z 492.333,A -85,B 0,C 180,E1 -2819.368,E2 -2819.368} C_VEL
LIN {X 0,Y 558.808,Z 495.074,A -85,B 0,C 180,E1 -2820.201,E2 -2820.201} C_VEL
LIN {X 0,Y 558.766,Z 497.374,A -85,B 0,C 180,E1 -2821.209,E2 -2821.209} C_VEL
LIN {X 0,Y 558.744,Z 498.32,A -85,B 0,C 180,E1 -2821.887,E2 -2821.887} C_VEL
LIN {X 0,Y 558.749,Z 498.893,A -85,B 0,C 180,E1 -2822.739,E2 -2822.739} C_VEL
LIN {X 0,Y 558.76,Z 498.642,A -85,B 0,C 180,E1 -2823.888,E2 -2823.888} C_VEL
LIN {X 0,Y 558.759,Z 496.814,A -85,B 0,C 180,E1 -2825.159,E2 -2825.159} C_VEL
LIN {X 0,Y 558.846,Z 494.012,A -85,B 0,C 180,E1 -2826.23,E2 -2826.23} C_VEL
LIN {X 0,Y 558.836,Z 490.697,A -85,B 0,C 180,E1 -2827.129,E2 -2827.129} C_VEL
LIN {X 0,Y 558.887,Z 486.354,A -85,B 0,C 180,E1 -2828.034,E2 -2828.034} C_VEL
LIN {X 0,Y 558.912,Z 480.737,A -85,B 0,C 180,E1 -2828.953,E2 -2828.953} C_VEL
LIN {X 0,Y 559.02,Z 473.614,A -85,B 0,C 180,E1 -2829.876,E2 -2829.876} C_VEL
LIN {X 0,Y 559.085,Z 465.71,A -85,B 0,C 180,E1 -2830.696,E2 -2830.696} C_VEL
LIN {X 0,Y 559.19,Z 456.309,A -85,B 0,C 180,E1 -2831.469,E2 -2831.469} C_VEL
LIN {X 0,Y 559.331,Z 445.345,A -85,B 0,C 180,E1 -2832.155,E2 -2832.155} C_VEL
LIN {X 0,Y 559.436,Z 437.054,A -85,B 0,C 180,E1 -2832.556,E2 -2832.556} C_VEL
LIN {X 0,Y 559.536,Z 426.721,A -85,B 0,C 180,E1 -2832.925,E2 -2832.925} C_VEL
LIN {X 0,Y 558.809,Z 419.331,A -85,B 0,C 180,E1 -2833.152,E2 -2833.152} C_VEL
LIN {X 0,Y 558.839,Z 412.295,A -85,B 0,C 180,E1 -2836.237,E2 -2836.237} C_VEL
LIN {X 0,Y 558.852,Z 405.707,A -85,B 0,C 180,E1 -2839.161,E2 -2839.161} C_VEL
LIN {X 0,Y 558.879,Z 399.526,A -85,B 0,C 180,E1 -2841.962,E2 -2841.962} C_VEL
LIN {X 0,Y 558.922,Z 393.378,A -85,B 0,C 180,E1 -2844.813,E2 -2844.813} C_VEL
LIN {X 0,Y 558.993,Z 387.968,A -85,B 0,C 180,E1 -2847.386,E2 -2847.386} C_VEL
LIN {X 0,Y 559.048,Z 382.282,A -85,B 0,C 180,E1 -2850.155,E2 -2850.155} C_VEL
LIN {X 0,Y 559.107,Z 377.783,A -85,B 0,C 180,E1 -2852.284,E2 -2852.284} C_VEL
LIN {X 0,Y 559.19,Z 372.531,A -85,B 0,C 180,E1 -2854.804,E2 -2854.804} C_VEL
LIN {X 0,Y 559.2,Z 370.831,A -85,B 0,C 180,E1 -2855.695,E2 -2855.695} C_VEL
LIN {X 0,Y 559.155,Z 370.835,A -85,B 0,C 180,E1 -2858.623,E2 -2858.623} C_VEL
LIN {X 0,Y 559.152,Z 370.837,A -85,B 0,C 180,E1 -2860.926,E2 -2860.926} C_VEL
LIN {X 0,Y 559.151,Z 370.836,A -85,B 0,C 180,E1 -2863.948,E2 -2863.948} C_VEL
LIN {X 0,Y 559.163,Z 370.836,A -85,B 0,C 180,E1 -2866.184,E2 -2866.184} C_VEL
LIN {X 0,Y 559.235,Z 370.825,A -85,B 0,C 180,E1 -2869.135,E2 -2869.135} C_VEL
LIN {X 0,Y 559.191,Z 370.83,A -85,B 0,C 180,E1 -2872.054,E2 -2872.054} C_VEL
LIN {X 0,Y 559.245,Z 370.824,A -85,B 0,C 180,E1 -2874.953,E2 -2874.953} C_VEL
LIN {X 0,Y 559.241,Z 370.827,A -85,B 0,C 180,E1 -2877.84,E2 -2877.84} C_VEL
LIN {X 0,Y 559.261,Z 370.824,A -85,B 0,C 180,E1 -2880.72,E2 -2880.72} C_VEL
LIN {X 0,Y 559.226,Z 370.826,A -85,B 0,C 180,E1 -2882.882,E2 -2882.882} C_VEL
LIN {X 0,Y 559.225,Z 370.828,A -85,B 0,C 180,E1 -2885.77,E2 -2885.77} C_VEL
LIN {X 0,Y 559.184,Z 370.834,A -85,B 0,C 180,E1 -2888.675,E2 -2888.675} C_VEL
LIN {X 0,Y 559.191,Z 370.831,A -85,B 0,C 180,E1 -2891.601,E2 -2891.601} C_VEL
LIN {X 0,Y 559.174,Z 370.832,A -85,B 0,C 180,E1 -2894.596,E2 -2894.596} C_VEL
LIN {X 0,Y 559.189,Z 370.831,A -85,B 0,C 180,E1 -2897.556,E2 -2897.556} C_VEL
LIN {X 0,Y 559.167,Z 370.837,A -85,B 0,C 180,E1 -2900.605,E2 -2900.605} C_VEL
LIN {X 0,Y 559.145,Z 370.836,A -85,B 0,C 180,E1 -2903.717,E2 -2903.717} C_VEL
LIN {X 0,Y 559.18,Z 370.834,A -85,B 0,C 180,E1 -2906.097,E2 -2906.097} C_VEL
LIN {X 0,Y 559.146,Z 370.838,A -85,B 0,C 180,E1 -2908.531,E2 -2908.531} C_VEL
LIN {X 0,Y 559.139,Z 370.84,A -85,B 0,C 180,E1 -2911.277,E2 -2911.277} C_VEL
LIN {X 0,Y 559.161,Z 370.837,A -85,B 0,C 180,E1 -2913.953,E2 -2913.953} C_VEL
LIN {X 0,Y 559.151,Z 370.836,A -85,B 0,C 180,E1 -2916.45,E2 -2916.45} C_VEL
LIN {X 0,Y 559.163,Z 370.834,A -85,B 0,C 180,E1 -2918.935,E2 -2918.935} C_VEL
LIN {X 0,Y 559.18,Z 370.833,A -85,B 0,C 180,E1 -2921.769,E2 -2921.769} C_VEL
LIN {X 0,Y 559.125,Z 370.842,A -85,B 0,C 180,E1 -2924.741,E2 -2924.741} C_VEL
LIN {X 0,Y 559.151,Z 370.838,A -85,B 0,C 180,E1 -2927.259,E2 -2927.259} C_VEL
LIN {X 0,Y 559.174,Z 370.836,A -85,B 0,C 180,E1 -2930.137,E2 -2930.137} C_VEL
LIN {X 0,Y 559.137,Z 370.84,A -85,B 0,C 180,E1 -2932.894,E2 -2932.894} C_VEL
LIN {X 0,Y 559.154,Z 370.839,A -85,B 0,C 180,E1 -2935.559,E2 -2935.559} C_VEL
LIN {X 0,Y 559.164,Z 370.837,A -85,B 0,C 180,E1 -2938.592,E2 -2938.592} C_VEL
LIN {X 0,Y 560.048,Z 375.849,A -85,B 0,C 180,E1 -2939.983,E2 -2939.983} C_VEL
LIN {X 0,Y 559.857,Z 386.836,A -85,B 0,C 180,E1 -2942.732,E2 -2942.732} C_VEL
LIN {X 0,Y 559.582,Z 398.317,A -85,B 0,C 180,E1 -2945.517,E2 -2945.517} C_VEL
LIN {X 0,Y 559.465,Z 410.955,A -85,B 0,C 180,E1 -2948.371,E2 -2948.371} C_VEL
LIN {X 0,Y 559.307,Z 423.904,A -85,B 0,C 180,E1 -2951.314,E2 -2951.314} C_VEL
LIN {X 0,Y 559.189,Z 435.68,A -85,B 0,C 180,E1 -2953.951,E2 -2953.951} C_VEL
LIN {X 0,Y 559.078,Z 447.456,A -85,B 0,C 180,E1 -2956.554,E2 -2956.554} C_VEL
LIN {X 0,Y 559.022,Z 450.085,A -85,B 0,C 180,E1 -2957.131,E2 -2957.131} C_VEL
LIN {X 0,Y 560.039,Z 457.323,A -85,B 0,C 180,E1 -2957.293,E2 -2957.293} C_VEL
LIN {X 0,Y 559.933,Z 470.556,A -85,B 0,C 180,E1 -2957.636,E2 -2957.636} C_VEL
LIN {X 0,Y 559.755,Z 482.559,A -85,B 0,C 180,E1 -2958.092,E2 -2958.092} C_VEL
LIN {X 0,Y 559.579,Z 494.631,A -85,B 0,C 180,E1 -2958.707,E2 -2958.707} C_VEL
LIN {X 0,Y 559.426,Z 505.51,A -85,B 0,C 180,E1 -2959.415,E2 -2959.415} C_VEL
LIN {X 0,Y 559.297,Z 515.667,A -85,B 0,C 180,E1 -2960.235,E2 -2960.235} C_VEL
LIN {X 0,Y 559.133,Z 524.803,A -85,B 0,C 180,E1 -2961.144,E2 -2961.144} C_VEL
LIN {X 0,Y 559.008,Z 533.702,A -85,B 0,C 180,E1 -2962.234,E2 -2962.234} C_VEL
LIN {X 0,Y 558.923,Z 539.752,A -85,B 0,C 180,E1 -2963.142,E2 -2963.142} C_VEL
LIN {X 0,Y 558.935,Z 545.688,A -85,B 0,C 180,E1 -2964.229,E2 -2964.229} C_VEL
LIN {X 0,Y 558.826,Z 550.378,A -85,B 0,C 180,E1 -2965.313,E2 -2965.313} C_VEL
LIN {X 0,Y 558.836,Z 553.964,A -85,B 0,C 180,E1 -2966.397,E2 -2966.397} C_VEL
LIN {X 0,Y 558.799,Z 555.814,A -85,B 0,C 180,E1 -2967.118,E2 -2967.118} C_VEL
LIN {X 0,Y 558.745,Z 558.188,A -85,B 0,C 180,E1 -2968.56,E2 -2968.56} C_VEL
LIN {X 0,Y 558.74,Z 559,A -85,B 0,C 180,E1 -2970.002,E2 -2970.002} C_VEL
LIN {X 0,Y 558.745,Z 558.183,A -85,B 0,C 180,E1 -2971.443,E2 -2971.443} C_VEL
LIN {X 0,Y 558.799,Z 555.804,A -85,B 0,C 180,E1 -2972.885,E2 -2972.885} C_VEL
LIN {X 0,Y 558.844,Z 552.89,A -85,B 0,C 180,E1 -2973.968,E2 -2973.968} C_VEL
LIN {X 0,Y 558.798,Z 548.944,A -85,B 0,C 180,E1 -2975.052,E2 -2975.052} C_VEL
LIN {X 0,Y 558.922,Z 543.86,A -85,B 0,C 180,E1 -2976.137,E2 -2976.137} C_VEL
LIN {X 0,Y 558.979,Z 537.458,A -85,B 0,C 180,E1 -2977.224,E2 -2977.224} C_VEL
LIN {X 0,Y 559.098,Z 529.466,A -85,B 0,C 180,E1 -2978.313,E2 -2978.313} C_VEL
LIN {X 0,Y 559.196,Z 521.321,A -85,B 0,C 180,E1 -2979.222,E2 -2979.222} C_VEL
LIN {X 0,Y 559.348,Z 511.384,A -85,B 0,C 180,E1 -2980.133,E2 -2980.133} C_VEL
LIN {X 0,Y 559.539,Z 500.404,A -85,B 0,C 180,E1 -2980.936,E2 -2980.936} C_VEL
LIN {X 0,Y 559.639,Z 488.793,A -85,B 0,C 180,E1 -2981.611,E2 -2981.611} C_VEL
LIN {X 0,Y 559.817,Z 476.956,A -85,B 0,C 180,E1 -2982.14,E2 -2982.14} C_VEL
LIN {X 0,Y 559.994,Z 464.13,A -85,B 0,C 180,E1 -2982.55,E2 -2982.55} C_VEL
LIN {X 0,Y 559.892,Z 455.309,A -85,B 0,C 180,E1 -2982.751,E2 -2982.751} C_VEL
LIN {X 0,Y 559.025,Z 450.07,A -85,B 0,C 180,E1 -2982.872,E2 -2982.872} C_VEL
LIN {X 0,Y 559.132,Z 439.03,A -85,B 0,C 180,E1 -2985.306,E2 -2985.306} C_VEL
LIN {X 0,Y 559.274,Z 427.254,A -85,B 0,C 180,E1 -2987.932,E2 -2987.932} C_VEL
LIN {X 0,Y 559.404,Z 415.478,A -85,B 0,C 180,E1 -2990.597,E2 -2990.597} C_VEL
LIN {X 0,Y 559.552,Z 403.978,A -85,B 0,C 180,E1 -2993.224,E2 -2993.224} C_VEL
LIN {X 0,Y 559.732,Z 391.705,A -85,B 0,C 180,E1 -2996.071,E2 -2996.071} C_VEL
LIN {X 0,Y 559.979,Z 380.228,A -85,B 0,C 180,E1 -2998.895,E2 -2998.895} C_VEL
LIN {X 0,Y 559.962,Z 375.298,A -85,B 0,C 180,E1 -3000.136,E2 -3000.136} C_VEL
LIN {X 0,Y 559.171,Z 370.835,A -85,B 0,C 180,E1 -3001.367,E2 -3001.367} C_VEL
LIN {X 0,Y 559.15,Z 370.837,A -85,B 0,C 180,E1 -3004.445,E2 -3004.445} C_VEL
LIN {X 0,Y 559.14,Z 370.835,A -85,B 0,C 180,E1 -3007.639,E2 -3007.639} C_VEL
LIN {X 0,Y 559.165,Z 370.837,A -85,B 0,C 180,E1 -3009.942,E2 -3009.942} C_VEL
LIN {X 0,Y 559.098,Z 370.841,A -85,B 0,C 180,E1 -3013.191,E2 -3013.191} C_VEL
LIN {X 0,Y 559.125,Z 370.836,A -85,B 0,C 180,E1 -3015.765,E2 -3015.765} C_VEL
LIN {X 0,Y 559.13,Z 370.834,A -85,B 0,C 180,E1 -3018.226,E2 -3018.226} C_VEL
LIN {X 0,Y 559.177,Z 370.829,A -85,B 0,C 180,E1 -3021.192,E2 -3021.192} C_VEL
LIN {X 0,Y 559.144,Z 370.833,A -85,B 0,C 180,E1 -3023.789,E2 -3023.789} C_VEL
LIN {X 0,Y 559.153,Z 370.835,A -85,B 0,C 180,E1 -3026.424,E2 -3026.424} C_VEL
LIN {X 0,Y 559.154,Z 370.831,A -85,B 0,C 180,E1 -3028.98,E2 -3028.98} C_VEL
LIN {X 0,Y 559.117,Z 370.842,A -85,B 0,C 180,E1 -3031.63,E2 -3031.63} C_VEL
LIN {X 0,Y 559.117,Z 370.836,A -85,B 0,C 180,E1 -3033.899,E2 -3033.899} C_VEL
LIN {X 0,Y 559.119,Z 370.841,A -85,B 0,C 180,E1 -3037.066,E2 -3037.066} C_VEL
LIN {X 0,Y 559.178,Z 370.828,A -85,B 0,C 180,E1 -3039.395,E2 -3039.395} C_VEL
LIN {X 0,Y 559.145,Z 370.833,A -85,B 0,C 180,E1 -3041.685,E2 -3041.685} C_VEL
LIN {X 0,Y 559.168,Z 370.836,A -85,B 0,C 180,E1 -3043.948,E2 -3043.948} C_VEL
LIN {X 0,Y 559.171,Z 370.833,A -85,B 0,C 180,E1 -3046.184,E2 -3046.184} C_VEL
LIN {X 0,Y 559.184,Z 370.832,A -85,B 0,C 180,E1 -3049.133,E2 -3049.133} C_VEL
LIN {X 0,Y 559.137,Z 370.834,A -85,B 0,C 180,E1 -3052.052,E2 -3052.052} C_VEL
LIN {X 0,Y 559.24,Z 370.827,A -85,B 0,C 180,E1 -3054.953,E2 -3054.953} C_VEL
LIN {X 0,Y 558.988,Z 371.01,A -85,B 0,C 180,E1 -3056.937,E2 -3056.937} C_VEL
LIN {X 0,Y 559.099,Z 379.122,A -85,B 0,C 180,E1 -3060,E2 -3060} C_VEL
LIN {X 0,Y 559.009,Z 386.49,A -85,B 0,C 180,E1 -3062.882,E2 -3062.882} C_VEL
LIN {X 0,Y 559.089,Z 391.858,A -85,B 0,C 180,E1 -3065.048,E2 -3065.048} C_VEL
LIN {X 0,Y 559.001,Z 398.805,A -85,B 0,C 180,E1 -3067.949,E2 -3067.949} C_VEL
LIN {X 0,Y 558.969,Z 405.813,A -85,B 0,C 180,E1 -3070.871,E2 -3070.871} C_VEL
LIN {X 0,Y 558.906,Z 412.82,A -85,B 0,C 180,E1 -3073.822,E2 -3073.822} C_VEL
LIN {X 0,Y 558.85,Z 420.031,A -85,B 0,C 180,E1 -3076.812,E2 -3076.812} C_VEL
LIN {X 0,Y 558.846,Z 423.481,A -85,B 0,C 180,E1 -3078.229,E2 -3078.229} C_VEL
LIN {X 0,Y 559.99,Z 431.416,A -85,B 0,C 180,E1 -3078.427,E2 -3078.427} C_VEL
LIN {X 0,Y 559.865,Z 442.917,A -85,B 0,C 180,E1 -3078.764,E2 -3078.764} C_VEL
LIN {X 0,Y 559.691,Z 453.916,A -85,B 0,C 180,E1 -3079.204,E2 -3079.204} C_VEL
LIN {X 0,Y 559.572,Z 464.586,A -85,B 0,C 180,E1 -3079.748,E2 -3079.748} C_VEL
LIN {X 0,Y 559.404,Z 476.036,A -85,B 0,C 180,E1 -3080.5,E2 -3080.5} C_VEL
LIN {X 0,Y 559.26,Z 487.881,A -85,B 0,C 180,E1 -3081.487,E2 -3081.487} C_VEL
LIN {X 0,Y 559.113,Z 496.191,A -85,B 0,C 180,E1 -3082.348,E2 -3082.348} C_VEL
LIN {X 0,Y 559.045,Z 502.802,A -85,B 0,C 180,E1 -3083.162,E2 -3083.162} C_VEL
LIN {X 0,Y 558.943,Z 509.306,A -85,B 0,C 180,E1 -3084.12,E2 -3084.12} C_VEL
LIN {X 0,Y 558.861,Z 514.871,A -85,B 0,C 180,E1 -3085.116,E2 -3085.116} C_VEL
LIN {X 0,Y 558.864,Z 515.801,A -85,B 0,C 180,E1 -3085.305,E2 -3085.305} C_VEL
LIN {X 0,Y 558.207,Z 518.357,A -85,B 0,C 180,E1 -3085.849,E2 -3085.849} C_VEL
LIN {X 0,Y 555.316,Z 521.91,A -85,B 0,C 180,E1 -3086.754,E2 -3086.754} C_VEL
LIN {X 0,Y 552.855,Z 524.218,A -85,B 0,C 180,E1 -3087.502,E2 -3087.502} C_VEL
LIN {X 0,Y 551.784,Z 525.689,A -85,B 0,C 180,E1 -3088.09,E2 -3088.09} C_VEL
LIN {X 0,Y 551.69,Z 526.098,A -85,B 0,C 180,E1 -3088.29,E2 -3088.29} C_VEL
LIN {X 0,Y 551.66,Z 527.357,A -85,B 0,C 180,E1 -3088.954,E2 -3088.954} C_VEL
LIN {X 0,Y 551.69,Z 528.569,A -85,B 0,C 180,E1 -3089.973,E2 -3089.973} C_VEL
LIN {X 0,Y 551.653,Z 528.931,A -85,B 0,C 180,E1 -3091.397,E2 -3091.397} C_VEL
LIN {X 0,Y 551.679,Z 527.887,A -85,B 0,C 180,E1 -3092.775,E2 -3092.775} C_VEL
LIN {X 0,Y 551.694,Z 525.479,A -85,B 0,C 180,E1 -3094.102,E2 -3094.102} C_VEL
LIN {X 0,Y 551.726,Z 521.82,A -85,B 0,C 180,E1 -3095.388,E2 -3095.388} C_VEL
LIN {X 0,Y 551.808,Z 516.874,A -85,B 0,C 180,E1 -3096.64,E2 -3096.64} C_VEL
LIN {X 0,Y 551.826,Z 510.61,A -85,B 0,C 180,E1 -3097.849,E2 -3097.849} C_VEL
LIN {X 0,Y 551.962,Z 502.766,A -85,B 0,C 180,E1 -3099.04,E2 -3099.04} C_VEL
LIN {X 0,Y 552.077,Z 494.896,A -85,B 0,C 180,E1 -3100.006,E2 -3100.006} C_VEL
LIN {X 0,Y 552.246,Z 485.488,A -85,B 0,C 180,E1 -3100.95,E2 -3100.95} C_VEL
LIN {X 0,Y 552.407,Z 475.249,A -85,B 0,C 180,E1 -3101.785,E2 -3101.785} C_VEL
LIN {X 0,Y 552.572,Z 463.565,A -85,B 0,C 180,E1 -3102.548,E2 -3102.548} C_VEL
LIN {X 0,Y 552.774,Z 451.047,A -85,B 0,C 180,E1 -3103.171,E2 -3103.171} C_VEL
LIN {X 0,Y 552.959,Z 438.106,A -85,B 0,C 180,E1 -3103.645,E2 -3103.645} C_VEL
LIN {X 0,Y 552.854,Z 430.082,A -85,B 0,C 180,E1 -3103.861,E2 -3103.861} C_VEL
LIN {X 0,Y 551.75,Z 423.459,A -85,B 0,C 180,E1 -3104.037,E2 -3104.037} C_VEL
LIN {X 0,Y 551.78,Z 416.251,A -85,B 0,C 180,E1 -3107.048,E2 -3107.048} C_VEL
LIN {X 0,Y 551.819,Z 409.69,A -85,B 0,C 180,E1 -3109.832,E2 -3109.832} C_VEL
LIN {X 0,Y 551.87,Z 402.733,A -85,B 0,C 180,E1 -3112.777,E2 -3112.777} C_VEL
LIN {X 0,Y 551.931,Z 397.481,A -85,B 0,C 180,E1 -3115.039,E2 -3115.039} C_VEL
LIN {X 0,Y 551.994,Z 390.261,A -85,B 0,C 180,E1 -3118.103,E2 -3118.103} C_VEL
LIN {X 0,Y 551.979,Z 383.303,A -85,B 0,C 180,E1 -3121.063,E2 -3121.063} C_VEL
LIN {X 0,Y 551.979,Z 377.373,A -85,B 0,C 180,E1 -3123.535,E2 -3123.535} C_VEL
LIN {X 0,Y 552.115,Z 371.714,A -85,B 0,C 180,E1 -3125.961,E2 -3125.961} C_VEL
LIN {X 0,Y 552.119,Z 371.712,A -85,B 0,C 180,E1 -3129.119,E2 -3129.119} C_VEL
LIN {X 0,Y 552.086,Z 371.714,A -85,B 0,C 180,E1 -3131.442,E2 -3131.442} C_VEL
LIN {X 0,Y 552.115,Z 371.714,A -85,B 0,C 180,E1 -3133.736,E2 -3133.736} C_VEL
LIN {X 0,Y 552.137,Z 371.707,A -85,B 0,C 180,E1 -3136.003,E2 -3136.003} C_VEL
LIN {X 0,Y 552.161,Z 371.704,A -85,B 0,C 180,E1 -3138.992,E2 -3138.992} C_VEL
LIN {X 0,Y 552.159,Z 371.705,A -85,B 0,C 180,E1 -3141.95,E2 -3141.95} C_VEL
LIN {X 0,Y 552.217,Z 371.7,A -85,B 0,C 180,E1 -3144.887,E2 -3144.887} C_VEL
LIN {X 0,Y 552.222,Z 371.702,A -85,B 0,C 180,E1 -3147.81,E2 -3147.81} C_VEL
LIN {X 0,Y 552.235,Z 371.767,A -85,B 0,C 180,E1 -3150.454,E2 -3150.454} C_VEL
LIN {X 0,Y 552.089,Z 376.771,A -85,B 0,C 180,E1 -3152.917,E2 -3152.917} C_VEL
LIN {X 0,Y 552.06,Z 382.751,A -85,B 0,C 180,E1 -3155.844,E2 -3155.844} C_VEL
LIN {X 0,Y 551.969,Z 388.905,A -85,B 0,C 180,E1 -3158.787,E2 -3158.787} C_VEL
LIN {X 0,Y 551.948,Z 394.272,A -85,B 0,C 180,E1 -3161.35,E2 -3161.35} C_VEL
LIN {X 0,Y 551.853,Z 401.543,A -85,B 0,C 180,E1 -3164.754,E2 -3164.754} C_VEL
LIN {X 0,Y 551.734,Z 408.104,A -85,B 0,C 180,E1 -3167.799,E2 -3167.799} C_VEL
LIN {X 0,Y 551.7,Z 413.271,A -85,B 0,C 180,E1 -3170.115,E2 -3170.115} C_VEL
LIN {X 0,Y 551.702,Z 419.342,A -85,B 0,C 180,E1 -3172.811,E2 -3172.811} C_VEL
LIN {X 0,Y 552.528,Z 427.025,A -85,B 0,C 180,E1 -3173.047,E2 -3173.047} C_VEL
LIN {X 0,Y 552.37,Z 438.721,A -85,B 0,C 180,E1 -3173.482,E2 -3173.482} C_VEL
LIN {X 0,Y 552.222,Z 449.068,A -85,B 0,C 180,E1 -3174.03,E2 -3174.03} C_VEL
LIN {X 0,Y 552.126,Z 457.909,A -85,B 0,C 180,E1 -3174.635,E2 -3174.635} C_VEL
LIN {X 0,Y 552.054,Z 466.035,A -85,B 0,C 180,E1 -3175.328,E2 -3175.328} C_VEL
LIN {X 0,Y 551.924,Z 473.025,A -85,B 0,C 180,E1 -3176.057,E2 -3176.057} C_VEL
LIN {X 0,Y 551.871,Z 479.923,A -85,B 0,C 180,E1 -3176.946,E2 -3176.946} C_VEL
LIN {X 0,Y 551.792,Z 485.869,A -85,B 0,C 180,E1 -3177.907,E2 -3177.907} C_VEL
LIN {X 0,Y 551.734,Z 490.864,A -85,B 0,C 180,E1 -3178.947,E2 -3178.947} C_VEL
LIN {X 0,Y 551.72,Z 494.521,A -85,B 0,C 180,E1 -3179.98,E2 -3179.98} C_VEL
LIN {X 0,Y 551.691,Z 496.193,A -85,B 0,C 180,E1 -3180.632,E2 -3180.632} C_VEL
LIN {X 0,Y 551.649,Z 497.794,A -85,B 0,C 180,E1 -3181.487,E2 -3181.487} C_VEL
LIN {X 0,Y 551.667,Z 498.909,A -85,B 0,C 180,E1 -3182.774,E2 -3182.774} C_VEL
LIN {X 0,Y 551.677,Z 498.472,A -85,B 0,C 180,E1 -3184.101,E2 -3184.101} C_VEL
LIN {X 0,Y 551.657,Z 497.253,A -85,B 0,C 180,E1 -3184.977,E2 -3184.977} C_VEL
LIN {X 0,Y 551.772,Z 494.088,A -85,B 0,C 180,E1 -3186.247,E2 -3186.247} C_VEL
LIN {X 0,Y 551.76,Z 490.492,A -85,B 0,C 180,E1 -3187.228,E2 -3187.228} C_VEL
LIN {X 0,Y 551.804,Z 485.779,A -85,B 0,C 180,E1 -3188.199,E2 -3188.199} C_VEL
LIN {X 0,Y 551.835,Z 480.754,A -85,B 0,C 180,E1 -3189.025,E2 -3189.025} C_VEL
LIN {X 0,Y 551.949,Z 474.205,A -85,B 0,C 180,E1 -3189.893,E2 -3189.893} C_VEL
LIN {X 0,Y 552.028,Z 467.645,A -85,B 0,C 180,E1 -3190.605,E2 -3190.605} C_VEL
LIN {X 0,Y 552.111,Z 459.585,A -85,B 0,C 180,E1 -3191.321,E2 -3191.321} C_VEL
LIN {X 0,Y 552.243,Z 451.227,A -85,B 0,C 180,E1 -3191.919,E2 -3191.919} C_VEL
LIN {X 0,Y 552.353,Z 442.844,A -85,B 0,C 180,E1 -3192.401,E2 -3192.401} C_VEL
LIN {X 0,Y 552.464,Z 434.461,A -85,B 0,C 180,E1 -3192.78,E2 -3192.78} C_VEL
LIN {X 0,Y 552.473,Z 425.352,A -85,B 0,C 180,E1 -3193.092,E2 -3193.092} C_VEL
LIN {X 0,Y 551.733,Z 419.345,A -85,B 0,C 180,E1 -3193.276,E2 -3193.276} C_VEL
LIN {X 0,Y 551.761,Z 411.978,A -85,B 0,C 180,E1 -3196.551,E2 -3196.551} C_VEL
LIN {X 0,Y 551.757,Z 405.483,A -85,B 0,C 180,E1 -3199.488,E2 -3199.488} C_VEL
LIN {X 0,Y 551.832,Z 399.535,A -85,B 0,C 180,E1 -3202.316,E2 -3202.316} C_VEL
LIN {X 0,Y 551.855,Z 393.682,A -85,B 0,C 180,E1 -3205.035,E2 -3205.035} C_VEL
LIN {X 0,Y 551.928,Z 388.154,A -85,B 0,C 180,E1 -3207.669,E2 -3207.669} C_VEL
LIN {X 0,Y 552.017,Z 382.963,A -85,B 0,C 180,E1 -3210.23,E2 -3210.23} C_VEL
LIN {X 0,Y 552.11,Z 377.19,A -85,B 0,C 180,E1 -3213,E2 -3213} C_VEL
LIN {X 0,Y 552.177,Z 371.706,A -85,B 0,C 180,E1 -3215.716,E2 -3215.716} C_VEL
LIN {X 0,Y 552.1,Z 371.715,A -85,B 0,C 180,E1 -3218.337,E2 -3218.337} C_VEL
LIN {X 0,Y 552.135,Z 371.714,A -85,B 0,C 180,E1 -3220.674,E2 -3220.674} C_VEL
LIN {X 0,Y 552.1,Z 371.715,A -85,B 0,C 180,E1 -3223.737,E2 -3223.737} C_VEL
LIN {X 0,Y 552.126,Z 371.714,A -85,B 0,C 180,E1 -3226.004,E2 -3226.004} C_VEL
LIN {X 0,Y 552.191,Z 371.703,A -85,B 0,C 180,E1 -3228.994,E2 -3228.994} C_VEL
LIN {X 0,Y 552.143,Z 371.708,A -85,B 0,C 180,E1 -3231.952,E2 -3231.952} C_VEL
LIN {X 0,Y 552.219,Z 371.699,A -85,B 0,C 180,E1 -3234.889,E2 -3234.889} C_VEL
LIN {X 0,Y 552.211,Z 371.702,A -85,B 0,C 180,E1 -3237.812,E2 -3237.812} C_VEL
LIN {X 0,Y 552.23,Z 371.699,A -85,B 0,C 180,E1 -3240.729,E2 -3240.729} C_VEL
LIN {X 0,Y 552.192,Z 371.703,A -85,B 0,C 180,E1 -3242.918,E2 -3242.918} C_VEL
LIN {X 0,Y 552.194,Z 371.704,A -85,B 0,C 180,E1 -3245.844,E2 -3245.844} C_VEL
LIN {X 0,Y 552.153,Z 371.709,A -85,B 0,C 180,E1 -3248.786,E2 -3248.786} C_VEL
LIN {X 0,Y 552.144,Z 371.708,A -85,B 0,C 180,E1 -3251.751,E2 -3251.751} C_VEL
LIN {X 0,Y 552.114,Z 371.711,A -85,B 0,C 180,E1 -3254.749,E2 -3254.749} C_VEL
LIN {X 0,Y 552.121,Z 371.713,A -85,B 0,C 180,E1 -3257.788,E2 -3257.788} C_VEL
LIN {X 0,Y 552.114,Z 371.712,A -85,B 0,C 180,E1 -3260.102,E2 -3260.102} C_VEL
LIN {X 0,Y 552.094,Z 371.714,A -85,B 0,C 180,E1 -3262.451,E2 -3262.451} C_VEL
LIN {X 0,Y 552.135,Z 371.709,A -85,B 0,C 180,E1 -3265.352,E2 -3265.352} C_VEL
LIN {X 0,Y 552.107,Z 371.712,A -85,B 0,C 180,E1 -3268.099,E2 -3268.099} C_VEL
LIN {X 0,Y 552.096,Z 371.713,A -85,B 0,C 180,E1 -3270.61,E2 -3270.61} C_VEL
LIN {X 0,Y 552.11,Z 371.712,A -85,B 0,C 180,E1 -3273.186,E2 -3273.186} C_VEL
LIN {X 0,Y 552.096,Z 371.714,A -85,B 0,C 180,E1 -3275.843,E2 -3275.843} C_VEL
LIN {X 0,Y 552.111,Z 371.713,A -85,B 0,C 180,E1 -3279.064,E2 -3279.064} C_VEL
LIN {X 0,Y 552.126,Z 371.71,A -85,B 0,C 180,E1 -3281.446,E2 -3281.446} C_VEL
LIN {X 0,Y 552.082,Z 371.718,A -85,B 0,C 180,E1 -3284.534,E2 -3284.534} C_VEL
LIN {X 0,Y 552.117,Z 371.714,A -85,B 0,C 180,E1 -3287.586,E2 -3287.586} C_VEL
LIN {X 0,Y 552.123,Z 371.712,A -85,B 0,C 180,E1 -3290.475,E2 -3290.475} C_VEL
LIN {X 0,Y 552.104,Z 371.714,A -85,B 0,C 180,E1 -3293.318,E2 -3293.318} C_VEL
LIN {X 0,Y 552.132,Z 371.711,A -85,B 0,C 180,E1 -3295.942,E2 -3295.942} C_VEL
LIN {X 0,Y 552.161,Z 371.884,A -85,B 0,C 180,E1 -3298.45,E2 -3298.45} C_VEL
LIN {X 0,Y 553.058,Z 376.695,A -85,B 0,C 180,E1 -3299.782,E2 -3299.782} C_VEL
LIN {X 0,Y 552.954,Z 385.202,A -85,B 0,C 180,E1 -3301.951,E2 -3301.951} C_VEL
LIN {X 0,Y 552.659,Z 396.915,A -85,B 0,C 180,E1 -3304.861,E2 -3304.861} C_VEL
LIN {X 0,Y 552.499,Z 406.727,A -85,B 0,C 180,E1 -3307.174,E2 -3307.174} C_VEL
LIN {X 0,Y 552.346,Z 418.802,A -85,B 0,C 180,E1 -3309.909,E2 -3309.909} C_VEL
LIN {X 0,Y 552.213,Z 432.315,A -85,B 0,C 180,E1 -3312.981,E2 -3312.981} C_VEL
LIN {X 0,Y 552.049,Z 445.774,A -85,B 0,C 180,E1 -3316.004,E2 -3316.004} C_VEL
LIN {X 0,Y 551.978,Z 450.085,A -85,B 0,C 180,E1 -3316.964,E2 -3316.964} C_VEL
LIN {X 0,Y 553.075,Z 458.461,A -85,B 0,C 180,E1 -3317.153,E2 -3317.153} C_VEL
LIN {X 0,Y 552.988,Z 470.555,A -85,B 0,C 180,E1 -3317.478,E2 -3317.478} C_VEL
LIN {X 0,Y 552.808,Z 482.549,A -85,B 0,C 180,E1 -3317.94,E2 -3317.94} C_VEL
LIN {X 0,Y 552.621,Z 493.291,A -85,B 0,C 180,E1 -3318.484,E2 -3318.484} C_VEL
LIN {X 0,Y 552.478,Z 504.225,A -85,B 0,C 180,E1 -3319.187,E2 -3319.187} C_VEL
LIN {X 0,Y 552.303,Z 514.624,A -85,B 0,C 180,E1 -3320.018,E2 -3320.018} C_VEL
LIN {X 0,Y 552.13,Z 523.131,A -85,B 0,C 180,E1 -3320.847,E2 -3320.847} C_VEL
LIN {X 0,Y 552.012,Z 530.975,A -85,B 0,C 180,E1 -3321.767,E2 -3321.767} C_VEL
LIN {X 0,Y 551.888,Z 538.633,A -85,B 0,C 180,E1 -3322.869,E2 -3322.869} C_VEL
LIN {X 0,Y 551.867,Z 545.688,A -85,B 0,C 180,E1 -3324.154,E2 -3324.154} C_VEL
LIN {X 0,Y 551.725,Z 550.379,A -85,B 0,C 180,E1 -3325.252,E2 -3325.252} C_VEL
LIN {X 0,Y 551.75,Z 553.965,A -85,B 0,C 180,E1 -3326.35,E2 -3326.35} C_VEL
LIN {X 0,Y 551.723,Z 555.814,A -85,B 0,C 180,E1 -3327.081,E2 -3327.081} C_VEL
LIN {X 0,Y 551.645,Z 558.187,A -85,B 0,C 180,E1 -3328.542,E2 -3328.542} C_VEL
LIN {X 0,Y 551.64,Z 559,A -85,B 0,C 180,E1 -3330.002,E2 -3330.002} C_VEL
LIN {X 0,Y 551.645,Z 558.182,A -85,B 0,C 180,E1 -3331.462,E2 -3331.462} C_VEL
LIN {X 0,Y 551.724,Z 555.804,A -85,B 0,C 180,E1 -3332.922,E2 -3332.922} C_VEL
LIN {X 0,Y 551.764,Z 552.89,A -85,B 0,C 180,E1 -3334.019,E2 -3334.019} C_VEL
LIN {X 0,Y 551.724,Z 548.944,A -85,B 0,C 180,E1 -3335.117,E2 -3335.117} C_VEL
LIN {X 0,Y 551.825,Z 543.189,A -85,B 0,C 180,E1 -3336.341,E2 -3336.341} C_VEL
LIN {X 0,Y 551.928,Z 536.227,A -85,B 0,C 180,E1 -3337.501,E2 -3337.501} C_VEL
LIN {X 0,Y 552.079,Z 527.98,A -85,B 0,C 180,E1 -3338.604,E2 -3338.604} C_VEL
LIN {X 0,Y 552.202,Z 519.525,A -85,B 0,C 180,E1 -3339.525,E2 -3339.525} C_VEL
LIN {X 0,Y 552.399,Z 509.078,A -85,B 0,C 180,E1 -3340.447,E2 -3340.447} C_VEL
LIN {X 0,Y 552.596,Z 497.255,A -85,B 0,C 180,E1 -3341.281,E2 -3341.281} C_VEL
LIN {X 0,Y 552.75,Z 485.462,A -85,B 0,C 180,E1 -3341.925,E2 -3341.925} C_VEL
LIN {X 0,Y 552.935,Z 473.137,A -85,B 0,C 180,E1 -3342.433,E2 -3342.433} C_VEL
LIN {X 0,Y 553.064,Z 460.468,A -85,B 0,C 180,E1 -3342.803,E2 -3342.803} C_VEL
LIN {X 0,Y 552.935,Z 456.021,A -85,B 0,C 180,E1 -3342.9,E2 -3342.9} C_VEL
LIN {X 0,Y 551.98,Z 450.07,A -85,B 0,C 180,E1 -3343.04,E2 -3343.04} C_VEL
LIN {X 0,Y 552.134,Z 437.347,A -85,B 0,C 180,E1 -3345.884,E2 -3345.884} C_VEL
LIN {X 0,Y 552.27,Z 425.571,A -85,B 0,C 180,E1 -3348.552,E2 -3348.552} C_VEL
LIN {X 0,Y 552.474,Z 412.024,A -85,B 0,C 180,E1 -3351.649,E2 -3351.649} C_VEL
LIN {X 0,Y 552.695,Z 398.421,A -85,B 0,C 180,E1 -3354.812,E2 -3354.812} C_VEL
LIN {X 0,Y 552.976,Z 385.189,A -85,B 0,C 180,E1 -3358.051,E2 -3358.051} C_VEL
LIN {X 0,Y 553.152,Z 378.611,A -85,B 0,C 180,E1 -3359.704,E2 -3359.704} C_VEL
LIN {X 0,Y 552.202,Z 372.076,A -85,B 0,C 180,E1 -3361.455,E2 -3361.455} C_VEL
LIN {X 0,Y 552.124,Z 371.71,A -85,B 0,C 180,E1 -3361.674,E2 -3361.674} C_VEL
LIN {X 0,Y 552.14,Z 371.709,A -85,B 0,C 180,E1 -3364.171,E2 -3364.171} C_VEL
LIN {X 0,Y 552.105,Z 371.713,A -85,B 0,C 180,E1 -3366.748,E2 -3366.748} C_VEL
LIN {X 0,Y 552.133,Z 371.708,A -85,B 0,C 180,E1 -3369.528,E2 -3369.528} C_VEL
LIN {X 0,Y 552.085,Z 371.713,A -85,B 0,C 180,E1 -3372.431,E2 -3372.431} C_VEL
LIN {X 0,Y 552.076,Z 371.716,A -85,B 0,C 180,E1 -3375.56,E2 -3375.56} C_VEL
LIN {X 0,Y 552.08,Z 371.715,A -85,B 0,C 180,E1 -3378.55,E2 -3378.55} C_VEL
LIN {X 0,Y 552.12,Z 371.707,A -85,B 0,C 180,E1 -3381.411,E2 -3381.411} C_VEL
LIN {X 0,Y 552.091,Z 371.716,A -85,B 0,C 180,E1 -3384.156,E2 -3384.156} C_VEL
LIN {X 0,Y 552.112,Z 371.709,A -85,B 0,C 180,E1 -3386.814,E2 -3386.814} C_VEL
LIN {X 0,Y 552.097,Z 371.713,A -85,B 0,C 180,E1 -3389.39,E2 -3389.39} C_VEL
LIN {X 0,Y 552.063,Z 371.717,A -85,B 0,C 180,E1 -3391.899,E2 -3391.899} C_VEL
LIN {X 0,Y 552.065,Z 371.716,A -85,B 0,C 180,E1 -3394.671,E2 -3394.671} C_VEL
LIN {X 0,Y 552.091,Z 371.711,A -85,B 0,C 180,E1 -3397.549,E2 -3397.549} C_VEL
LIN {X 0,Y 552.148,Z 371.711,A -85,B 0,C 180,E1 -3400.375,E2 -3400.375} C_VEL
LIN {X 0,Y 552.159,Z 371.703,A -85,B 0,C 180,E1 -3402.977,E2 -3402.977} C_VEL
LIN {X 0,Y 552.137,Z 371.712,A -85,B 0,C 180,E1 -3406.004,E2 -3406.004} C_VEL
LIN {X 0,Y 552.156,Z 371.706,A -85,B 0,C 180,E1 -3408.993,E2 -3408.993} C_VEL
LIN {X 0,Y 552.107,Z 371.71,A -85,B 0,C 180,E1 -3411.951,E2 -3411.951} C_VEL
LIN {X 0,Y 552.215,Z 371.703,A -85,B 0,C 180,E1 -3414.889,E2 -3414.889} C_VEL
LIN {X 0,Y 551.92,Z 371.89,A -85,B 0,C 180,E1 -3416.989,E2 -3416.989} C_VEL
LIN {X 0,Y 552.052,Z 379.801,A -85,B 0,C 180,E1 -3420,E2 -3420} C_VEL
LIN {X 0,Y 551.935,Z 387.253,A -85,B 0,C 180,E1 -3422.919,E2 -3422.919} C_VEL
LIN {X 0,Y 552.014,Z 392.657,A -85,B 0,C 180,E1 -3425.113,E2 -3425.113} C_VEL
LIN {X 0,Y 551.939,Z 399.604,A -85,B 0,C 180,E1 -3428.051,E2 -3428.051} C_VEL
LIN {X 0,Y 551.91,Z 407.476,A -85,B 0,C 180,E1 -3431.328,E2 -3431.328} C_VEL
LIN {X 0,Y 551.821,Z 415.571,A -85,B 0,C 180,E1 -3434.757,E2 -3434.757} C_VEL
LIN {X 0,Y 551.726,Z 422.855,A -85,B 0,C 180,E1 -3437.801,E2 -3437.801} C_VEL
LIN {X 0,Y 551.734,Z 423.489,A -85,B 0,C 180,E1 -3438.064,E2 -3438.064} C_VEL
LIN {X 0,Y 553.047,Z 432.027,A -85,B 0,C 180,E1 -3438.284,E2 -3438.284} C_VEL
LIN {X 0,Y 552.934,Z 443.326,A -85,B 0,C 180,E1 -3438.623,E2 -3438.623} C_VEL
LIN {X 0,Y 552.73,Z 454.137,A -85,B 0,C 180,E1 -3439.063,E2 -3439.063} C_VEL
LIN {X 0,Y 552.632,Z 463.566,A -85,B 0,C 180,E1 -3439.544,E2 -3439.544} C_VEL
LIN {X 0,Y 552.446,Z 473.503,A -85,B 0,C 180,E1 -3440.186,E2 -3440.186} C_VEL
LIN {X 0,Y 552.334,Z 482.337,A -85,B 0,C 180,E1 -3440.871,E2 -3440.871} C_VEL
LIN {X 0,Y 552.178,Z 491.231,A -85,B 0,C 180,E1 -3441.7,E2 -3441.7} C_VEL
LIN {X 0,Y 552.046,Z 499.668,A -85,B 0,C 180,E1 -3442.65,E2 -3442.65} C_VEL
LIN {X 0,Y 551.915,Z 507.624,A -85,B 0,C 180,E1 -3443.754,E2 -3443.754} C_VEL
LIN {X 0,Y 551.827,Z 513.944,A -85,B 0,C 180,E1 -3444.852,E2 -3444.852} C_VEL
LIN {X 0,Y 551.756,Z 519.507,A -85,B 0,C 180,E1 -3446.068,E2 -3446.068} C_VEL
LIN {X 0,Y 551.724,Z 523.631,A -85,B 0,C 180,E1 -3447.295,E2 -3447.295} C_VEL
LIN {X 0,Y 551.69,Z 526.098,A -85,B 0,C 180,E1 -3448.29,E2 -3448.29} C_VEL
LIN {X 0,Y 550.996,Z 527.263,A -85,B 0,C 180,E1 -3448.889,E2 -3448.889} C_VEL
LIN {X 0,Y 548.096,Z 528.489,A -85,B 0,C 180,E1 -3449.87,E2 -3449.87} C_VEL
LIN {X 0,Y 545.662,Z 528.928,A -85,B 0,C 180,E1 -3450.665,E2 -3450.665} C_VEL
LIN {X 0,Y 544.625,Z 528.964,A -85,B 0,C 180,E1 -3451.28,E2 -3451.28} C_VEL
LIN {X 0,Y 544.544,Z 528.911,A -85,B 0,C 180,E1 -3451.488,E2 -3451.488} C_VEL
LIN {X 0,Y 544.578,Z 527.622,A -85,B 0,C 180,E1 -3452.98,E2 -3452.98} C_VEL
LIN {X 0,Y 544.609,Z 525.058,A -85,B 0,C 180,E1 -3454.319,E2 -3454.319} C_VEL
LIN {X 0,Y 544.635,Z 521.258,A -85,B 0,C 180,E1 -3455.613,E2 -3455.613} C_VEL
LIN {X 0,Y 544.738,Z 516.109,A -85,B 0,C 180,E1 -3456.879,E2 -3456.879} C_VEL
LIN {X 0,Y 544.786,Z 509.653,A -85,B 0,C 180,E1 -3458.1,E2 -3458.1} C_VEL
LIN {X 0,Y 544.95,Z 501.594,A -85,B 0,C 180,E1 -3459.303,E2 -3459.303} C_VEL
LIN {X 0,Y 545.096,Z 493.181,A -85,B 0,C 180,E1 -3460.31,E2 -3460.31} C_VEL
LIN {X 0,Y 545.273,Z 483.79,A -85,B 0,C 180,E1 -3461.231,E2 -3461.231} C_VEL
LIN {X 0,Y 545.454,Z 473.32,A -85,B 0,C 180,E1 -3462.067,E2 -3462.067} C_VEL
LIN {X 0,Y 545.624,Z 462.434,A -85,B 0,C 180,E1 -3462.76,E2 -3462.76} C_VEL
LIN {X 0,Y 545.839,Z 450.584,A -85,B 0,C 180,E1 -3463.348,E2 -3463.348} C_VEL
LIN {X 0,Y 546.044,Z 437.551,A -85,B 0,C 180,E1 -3463.824,E2 -3463.824} C_VEL
LIN {X 0,Y 545.925,Z 431.134,A -85,B 0,C 180,E1 -3464.001,E2 -3464.001} C_VEL
LIN {X 0,Y 544.669,Z 423.473,A -85,B 0,C 180,E1 -3464.204,E2 -3464.204} C_VEL
LIN {X 0,Y 544.698,Z 417.206,A -85,B 0,C 180,E1 -3466.855,E2 -3466.855} C_VEL
LIN {X 0,Y 544.75,Z 410.373,A -85,B 0,C 180,E1 -3469.828,E2 -3469.828} C_VEL
LIN {X 0,Y 544.788,Z 403.589,A -85,B 0,C 180,E1 -3472.675,E2 -3472.675} C_VEL
LIN {X 0,Y 544.864,Z 397.283,A -85,B 0,C 180,E1 -3475.42,E2 -3475.42} C_VEL
LIN {X 0,Y 544.941,Z 390.438,A -85,B 0,C 180,E1 -3478.341,E2 -3478.341} C_VEL
LIN {X 0,Y 544.942,Z 383.056,A -85,B 0,C 180,E1 -3481.497,E2 -3481.497} C_VEL
LIN {X 0,Y 544.963,Z 375.888,A -85,B 0,C 180,E1 -3484.52,E2 -3484.52} C_VEL
LIN {X 0,Y 545.071,Z 372.591,A -85,B 0,C 180,E1 -3485.988,E2 -3485.988} C_VEL
LIN {X 0,Y 545.066,Z 372.593,A -85,B 0,C 180,E1 -3488.835,E2 -3488.835} C_VEL
LIN {X 0,Y 545.051,Z 372.59,A -85,B 0,C 180,E1 -3491.193,E2 -3491.193} C_VEL
LIN {X 0,Y 545.066,Z 372.593,A -85,B 0,C 180,E1 -3493.52,E2 -3493.52} C_VEL
LIN {X 0,Y 545.097,Z 372.584,A -85,B 0,C 180,E1 -3495.819,E2 -3495.819} C_VEL
LIN {X 0,Y 545.118,Z 372.582,A -85,B 0,C 180,E1 -3498.848,E2 -3498.848} C_VEL
LIN {X 0,Y 545.129,Z 372.581,A -85,B 0,C 180,E1 -3501.846,E2 -3501.846} C_VEL
LIN {X 0,Y 545.194,Z 372.576,A -85,B 0,C 180,E1 -3504.821,E2 -3504.821} C_VEL
LIN {X 0,Y 545.193,Z 372.577,A -85,B 0,C 180,E1 -3507.782,E2 -3507.782} C_VEL
LIN {X 0,Y 545.208,Z 372.721,A -85,B 0,C 180,E1 -3510.46,E2 -3510.46} C_VEL
LIN {X 0,Y 545.182,Z 376.24,A -85,B 0,C 180,E1 -3512.215,E2 -3512.215} C_VEL
LIN {X 0,Y 545.018,Z 382.21,A -85,B 0,C 180,E1 -3515.177,E2 -3515.177} C_VEL
LIN {X 0,Y 544.941,Z 388.34,A -85,B 0,C 180,E1 -3518.154,E2 -3518.154} C_VEL
LIN {X 0,Y 544.881,Z 395.132,A -85,B 0,C 180,E1 -3521.403,E2 -3521.403} C_VEL
LIN {X 0,Y 544.823,Z 402.024,A -85,B 0,C 180,E1 -3524.655,E2 -3524.655} C_VEL
LIN {X 0,Y 544.711,Z 407.595,A -85,B 0,C 180,E1 -3527.3,E2 -3527.3} C_VEL
LIN {X 0,Y 544.62,Z 414.253,A -85,B 0,C 180,E1 -3530.388,E2 -3530.388} C_VEL
LIN {X 0,Y 544.609,Z 419.336,A -85,B 0,C 180,E1 -3532.674,E2 -3532.674} C_VEL
LIN {X 0,Y 545.542,Z 427.542,A -85,B 0,C 180,E1 -3532.933,E2 -3532.933} C_VEL
LIN {X 0,Y 545.37,Z 439.462,A -85,B 0,C 180,E1 -3533.393,E2 -3533.393} C_VEL
LIN {X 0,Y 545.197,Z 449.452,A -85,B 0,C 180,E1 -3533.938,E2 -3533.938} C_VEL
LIN {X 0,Y 545.081,Z 458.423,A -85,B 0,C 180,E1 -3534.568,E2 -3534.568} C_VEL
LIN {X 0,Y 545.01,Z 465.562,A -85,B 0,C 180,E1 -3535.182,E2 -3535.182} C_VEL
LIN {X 0,Y 544.854,Z 473.377,A -85,B 0,C 180,E1 -3536.01,E2 -3536.01} C_VEL
LIN {X 0,Y 544.809,Z 479.712,A -85,B 0,C 180,E1 -3536.837,E2 -3536.837} C_VEL
LIN {X 0,Y 544.692,Z 484.946,A -85,B 0,C 180,E1 -3537.675,E2 -3537.675} C_VEL
LIN {X 0,Y 544.658,Z 489.197,A -85,B 0,C 180,E1 -3538.515,E2 -3538.515} C_VEL
LIN {X 0,Y 544.673,Z 492.609,A -85,B 0,C 180,E1 -3539.359,E2 -3539.359} C_VEL
LIN {X 0,Y 544.626,Z 495.283,A -85,B 0,C 180,E1 -3540.214,E2 -3540.214} C_VEL
LIN {X 0,Y 544.56,Z 497.234,A -85,B 0,C 180,E1 -3541.077,E2 -3541.077} C_VEL
LIN {X 0,Y 544.552,Z 498.437,A -85,B 0,C 180,E1 -3541.945,E2 -3541.945} C_VEL
LIN {X 0,Y 544.564,Z 498.992,A -85,B 0,C 180,E1 -3542.979,E2 -3542.979} C_VEL
LIN {X 0,Y 544.577,Z 498.217,A -85,B 0,C 180,E1 -3544.316,E2 -3544.316} C_VEL
LIN {X 0,Y 544.587,Z 495.912,A -85,B 0,C 180,E1 -3545.608,E2 -3545.608} C_VEL
LIN {X 0,Y 544.663,Z 493.691,A -85,B 0,C 180,E1 -3546.407,E2 -3546.407} C_VEL
LIN {X 0,Y 544.697,Z 490.282,A -85,B 0,C 180,E1 -3547.328,E2 -3547.328} C_VEL
LIN {X 0,Y 544.741,Z 485.806,A -85,B 0,C 180,E1 -3548.26,E2 -3548.26} C_VEL
LIN {X 0,Y 544.775,Z 481.679,A -85,B 0,C 180,E1 -3548.967,E2 -3548.967} C_VEL
LIN {X 0,Y 544.886,Z 474.701,A -85,B 0,C 180,E1 -3549.921,E2 -3549.921} C_VEL
LIN {X 0,Y 544.961,Z 468.084,A -85,B 0,C 180,E1 -3550.659,E2 -3550.659} C_VEL
LIN {X 0,Y 545.071,Z 460.435,A -85,B 0,C 180,E1 -3551.358,E2 -3551.358} C_VEL
LIN {X 0,Y 545.201,Z 452.715,A -85,B 0,C 180,E1 -3551.936,E2 -3551.936} C_VEL
LIN {X 0,Y 545.329,Z 444.354,A -85,B 0,C 180,E1 -3552.442,E2 -3552.442} C_VEL
LIN {X 0,Y 545.445,Z 435.407,A -85,B 0,C 180,E1 -3552.868,E2 -3552.868} C_VEL
LIN {X 0,Y 545.495,Z 426.045,A -85,B 0,C 180,E1 -3553.201,E2 -3553.201} C_VEL
LIN {X 0,Y 544.631,Z 419.329,A -85,B 0,C 180,E1 -3553.419,E2 -3553.419} C_VEL
LIN {X 0,Y 544.683,Z 413.009,A -85,B 0,C 180,E1 -3556.263,E2 -3556.263} C_VEL
LIN {X 0,Y 544.7,Z 405.988,A -85,B 0,C 180,E1 -3559.57,E2 -3559.57} C_VEL
LIN {X 0,Y 544.773,Z 399.491,A -85,B 0,C 180,E1 -3562.675,E2 -3562.675} C_VEL
LIN {X 0,Y 544.811,Z 393.673,A -85,B 0,C 180,E1 -3565.418,E2 -3565.418} C_VEL
LIN {X 0,Y 544.904,Z 387.619,A -85,B 0,C 180,E1 -3568.342,E2 -3568.342} C_VEL
LIN {X 0,Y 545.032,Z 381.139,A -85,B 0,C 180,E1 -3571.504,E2 -3571.504} C_VEL
LIN {X 0,Y 545.136,Z 375.096,A -85,B 0,C 180,E1 -3574.476,E2 -3574.476} C_VEL
LIN {X 0,Y 545.132,Z 372.584,A -85,B 0,C 180,E1 -3575.732,E2 -3575.732} C_VEL
LIN {X 0,Y 545.047,Z 372.593,A -85,B 0,C 180,E1 -3578.836,E2 -3578.836} C_VEL
LIN {X 0,Y 545.066,Z 372.591,A -85,B 0,C 180,E1 -3581.195,E2 -3581.195} C_VEL
LIN {X 0,Y 545.055,Z 372.594,A -85,B 0,C 180,E1 -3583.521,E2 -3583.521} C_VEL
LIN {X 0,Y 545.081,Z 372.591,A -85,B 0,C 180,E1 -3585.82,E2 -3585.82} C_VEL
LIN {X 0,Y 545.136,Z 372.583,A -85,B 0,C 180,E1 -3588.85,E2 -3588.85} C_VEL
LIN {X 0,Y 545.113,Z 372.583,A -85,B 0,C 180,E1 -3591.847,E2 -3591.847} C_VEL
LIN {X 0,Y 545.194,Z 372.574,A -85,B 0,C 180,E1 -3594.823,E2 -3594.823} C_VEL
LIN {X 0,Y 545.182,Z 372.578,A -85,B 0,C 180,E1 -3597.784,E2 -3597.784} C_VEL
LIN {X 0,Y 545.199,Z 372.575,A -85,B 0,C 180,E1 -3600.739,E2 -3600.739} C_VEL
LIN {X 0,Y 545.157,Z 372.579,A -85,B 0,C 180,E1 -3602.956,E2 -3602.956} C_VEL
LIN {X 0,Y 545.165,Z 372.581,A -85,B 0,C 180,E1 -3605.92,E2 -3605.92} C_VEL
LIN {X 0,Y 545.11,Z 372.585,A -85,B 0,C 180,E1 -3608.9,E2 -3608.9} C_VEL
LIN {X 0,Y 545.114,Z 372.583,A -85,B 0,C 180,E1 -3611.905,E2 -3611.905} C_VEL
LIN {X 0,Y 545.063,Z 372.59,A -85,B 0,C 180,E1 -3614.944,E2 -3614.944} C_VEL
LIN {X 0,Y 545.121,Z 372.583,A -85,B 0,C 180,E1 -3617.447,E2 -3617.447} C_VEL
LIN {X 0,Y 545.078,Z 372.589,A -85,B 0,C 180,E1 -3620.373,E2 -3620.373} C_VEL
LIN {X 0,Y 545.046,Z 372.592,A -85,B 0,C 180,E1 -3622.758,E2 -3622.758} C_VEL
LIN {X 0,Y 545.078,Z 372.588,A -85,B 0,C 180,E1 -3625.512,E2 -3625.512} C_VEL
LIN {X 0,Y 545.085,Z 372.589,A -85,B 0,C 180,E1 -3628.494,E2 -3628.494} C_VEL
LIN {X 0,Y 545.051,Z 372.592,A -85,B 0,C 180,E1 -3631.049,E2 -3631.049} C_VEL
LIN {X 0,Y 545.06,Z 372.591,A -85,B 0,C 180,E1 -3633.673,E2 -3633.673} C_VEL
LIN {X 0,Y 545.038,Z 372.594,A -85,B 0,C 180,E1 -3636.381,E2 -3636.381} C_VEL
LIN {X 0,Y 545.091,Z 372.59,A -85,B 0,C 180,E1 -3639.326,E2 -3639.326} C_VEL
LIN {X 0,Y 545.068,Z 372.593,A -85,B 0,C 180,E1 -3642.104,E2 -3642.104} C_VEL
LIN {X 0,Y 545.049,Z 372.591,A -85,B 0,C 180,E1 -3645.169,E2 -3645.169} C_VEL
LIN {X 0,Y 545.07,Z 372.589,A -85,B 0,C 180,E1 -3647.9,E2 -3647.9} C_VEL
LIN {X 0,Y 545.094,Z 372.586,A -85,B 0,C 180,E1 -3650.678,E2 -3650.678} C_VEL
LIN {X 0,Y 545.046,Z 372.593,A -85,B 0,C 180,E1 -3653.623,E2 -3653.623} C_VEL
LIN {X 0,Y 545.069,Z 372.592,A -85,B 0,C 180,E1 -3656.331,E2 -3656.331} C_VEL
LIN {X 0,Y 545.113,Z 372.724,A -85,B 0,C 180,E1 -3658.202,E2 -3658.202} C_VEL
LIN {X 0,Y 546.162,Z 378.709,A -85,B 0,C 180,E1 -3659.88,E2 -3659.88} C_VEL
LIN {X 0,Y 545.955,Z 389.473,A -85,B 0,C 180,E1 -3662.652,E2 -3662.652} C_VEL
LIN {X 0,Y 545.6,Z 402.705,A -85,B 0,C 180,E1 -3665.956,E2 -3665.956} C_VEL
LIN {X 0,Y 545.403,Z 413.461,A -85,B 0,C 180,E1 -3668.471,E2 -3668.471} C_VEL
LIN {X 0,Y 545.212,Z 427.168,A -85,B 0,C 180,E1 -3671.592,E2 -3671.592} C_VEL
LIN {X 0,Y 545.074,Z 439.045,A -85,B 0,C 180,E1 -3674.292,E2 -3674.292} C_VEL
LIN {X 0,Y 544.929,Z 450.085,A -85,B 0,C 180,E1 -3676.792,E2 -3676.792} C_VEL
LIN {X 0,Y 546.161,Z 458.46,A -85,B 0,C 180,E1 -3676.988,E2 -3676.988} C_VEL
LIN {X 0,Y 546.047,Z 470.555,A -85,B 0,C 180,E1 -3677.316,E2 -3677.316} C_VEL
LIN {X 0,Y 545.863,Z 482.547,A -85,B 0,C 180,E1 -3677.784,E2 -3677.784} C_VEL
LIN {X 0,Y 545.635,Z 494.194,A -85,B 0,C 180,E1 -3678.389,E2 -3678.389} C_VEL
LIN {X 0,Y 545.47,Z 505.513,A -85,B 0,C 180,E1 -3679.141,E2 -3679.141} C_VEL
LIN {X 0,Y 545.28,Z 515.666,A -85,B 0,C 180,E1 -3679.982,E2 -3679.982} C_VEL
LIN {X 0,Y 545.08,Z 524.802,A -85,B 0,C 180,E1 -3680.914,E2 -3680.914} C_VEL
LIN {X 0,Y 544.915,Z 533.702,A -85,B 0,C 180,E1 -3682.032,E2 -3682.032} C_VEL
LIN {X 0,Y 544.783,Z 540.86,A -85,B 0,C 180,E1 -3683.148,E2 -3683.148} C_VEL
LIN {X 0,Y 544.741,Z 547.373,A -85,B 0,C 180,E1 -3684.449,E2 -3684.449} C_VEL
LIN {X 0,Y 544.66,Z 551.683,A -85,B 0,C 180,E1 -3685.561,E2 -3685.561} C_VEL
LIN {X 0,Y 544.669,Z 553.965,A -85,B 0,C 180,E1 -3686.303,E2 -3686.303} C_VEL
LIN {X 0,Y 544.65,Z 555.814,A -85,B 0,C 180,E1 -3687.043,E2 -3687.043} C_VEL
LIN {X 0,Y 544.546,Z 558.186,A -85,B 0,C 180,E1 -3688.523,E2 -3688.523} C_VEL
LIN {X 0,Y 544.541,Z 559,A -85,B 0,C 180,E1 -3690.002,E2 -3690.002} C_VEL
LIN {X 0,Y 544.546,Z 558.182,A -85,B 0,C 180,E1 -3691.481,E2 -3691.481} C_VEL
LIN {X 0,Y 544.651,Z 555.804,A -85,B 0,C 180,E1 -3692.96,E2 -3692.96} C_VEL
LIN {X 0,Y 544.684,Z 552.89,A -85,B 0,C 180,E1 -3694.071,E2 -3694.071} C_VEL
LIN {X 0,Y 544.654,Z 548.944,A -85,B 0,C 180,E1 -3695.184,E2 -3695.184} C_VEL
LIN {X 0,Y 544.738,Z 543.595,A -85,B 0,C 180,E1 -3696.349,E2 -3696.349} C_VEL
LIN {X 0,Y 544.861,Z 536.226,A -85,B 0,C 180,E1 -3697.599,E2 -3697.599} C_VEL
LIN {X 0,Y 545.027,Z 527.98,A -85,B 0,C 180,E1 -3698.716,E2 -3698.716} C_VEL
LIN {X 0,Y 545.166,Z 519.525,A -85,B 0,C 180,E1 -3699.649,E2 -3699.649} C_VEL
LIN {X 0,Y 545.396,Z 509.076,A -85,B 0,C 180,E1 -3700.582,E2 -3700.582} C_VEL
LIN {X 0,Y 545.621,Z 497.639,A -85,B 0,C 180,E1 -3701.402,E2 -3701.402} C_VEL
LIN {X 0,Y 545.767,Z 487.382,A -85,B 0,C 180,E1 -3701.986,E2 -3701.986} C_VEL
LIN {X 0,Y 545.947,Z 475.735,A -85,B 0,C 180,E1 -3702.501,E2 -3702.501} C_VEL
LIN {X 0,Y 546.149,Z 462.299,A -85,B 0,C 180,E1 -3702.921,E2 -3702.921} C_VEL
LIN {X 0,Y 545.885,Z 456.021,A -85,B 0,C 180,E1 -3703.069,E2 -3703.069} C_VEL
LIN {X 0,Y 544.931,Z 450.07,A -85,B 0,C 180,E1 -3703.211,E2 -3703.211} C_VEL
LIN {X 0,Y 545.108,Z 437.347,A -85,B 0,C 180,E1 -3706.094,E2 -3706.094} C_VEL
LIN {X 0,Y 545.26,Z 425.515,A -85,B 0,C 180,E1 -3708.799,E2 -3708.799} C_VEL
LIN {X 0,Y 545.477,Z 411.932,A -85,B 0,C 180,E1 -3711.941,E2 -3711.941} C_VEL
LIN {X 0,Y 545.736,Z 398.425,A -85,B 0,C 180,E1 -3715.15,E2 -3715.15} C_VEL
LIN {X 0,Y 546.018,Z 386.845,A -85,B 0,C 180,E1 -3718.023,E2 -3718.023} C_VEL
LIN {X 0,Y 546.127,Z 378.633,A -85,B 0,C 180,E1 -3720.126,E2 -3720.126} C_VEL
LIN {X 0,Y 545.097,Z 372.585,A -85,B 0,C 180,E1 -3721.802,E2 -3721.802} C_VEL
LIN {X 0,Y 545.069,Z 372.591,A -85,B 0,C 180,E1 -3724.565,E2 -3724.565} C_VEL
LIN {X 0,Y 545.037,Z 372.591,A -85,B 0,C 180,E1 -3727.305,E2 -3727.305} C_VEL
LIN {X 0,Y 545.064,Z 372.592,A -85,B 0,C 180,E1 -3730.144,E2 -3730.144} C_VEL
LIN {X 0,Y 545.003,Z 372.596,A -85,B 0,C 180,E1 -3733.115,E2 -3733.115} C_VEL
LIN {X 0,Y 545.034,Z 372.59,A -85,B 0,C 180,E1 -3735.868,E2 -3735.868} C_VEL
LIN {X 0,Y 545.034,Z 372.596,A -85,B 0,C 180,E1 -3738.881,E2 -3738.881} C_VEL
LIN {X 0,Y 545.083,Z 372.59,A -85,B 0,C 180,E1 -3740.818,E2 -3740.818} C_VEL
LIN {X 0,Y 545.047,Z 372.589,A -85,B 0,C 180,E1 -3743.62,E2 -3743.62} C_VEL
LIN {X 0,Y 545.055,Z 372.592,A -85,B 0,C 180,E1 -3746.327,E2 -3746.327} C_VEL
LIN {X 0,Y 545.067,Z 372.586,A -85,B 0,C 180,E1 -3748.952,E2 -3748.952} C_VEL
LIN {X 0,Y 545.045,Z 372.596,A -85,B 0,C 180,E1 -3751.504,E2 -3751.504} C_VEL
LIN {X 0,Y 545.011,Z 372.594,A -85,B 0,C 180,E1 -3754.511,E2 -3754.511} C_VEL
LIN {X 0,Y 545.035,Z 372.593,A -85,B 0,C 180,E1 -3757.242,E2 -3757.242} C_VEL
LIN {X 0,Y 545.12,Z 372.586,A -85,B 0,C 180,E1 -3760.415,E2 -3760.415} C_VEL
LIN {X 0,Y 545.075,Z 372.587,A -85,B 0,C 180,E1 -3763.521,E2 -3763.521} C_VEL
LIN {X 0,Y 545.097,Z 372.589,A -85,B 0,C 180,E1 -3765.82,E2 -3765.82} C_VEL
LIN {X 0,Y 545.114,Z 372.582,A -85,B 0,C 180,E1 -3768.849,E2 -3768.849} C_VEL
LIN {X 0,Y 545.065,Z 372.588,A -85,B 0,C 180,E1 -3771.846,E2 -3771.846} C_VEL
LIN {X 0,Y 545.191,Z 372.578,A -85,B 0,C 180,E1 -3774.823,E2 -3774.823} C_VEL
LIN {X 0,Y 544.859,Z 372.7,A -85,B 0,C 180,E1 -3776.996,E2 -3776.996} C_VEL
LIN {X 0,Y 545.007,Z 380.522,A -85,B 0,C 180,E1 -3780,E2 -3780} C_VEL
LIN {X 0,Y 544.865,Z 386.172,A -85,B 0,C 180,E1 -3782.217,E2 -3782.217} C_VEL
LIN {X 0,Y 544.944,Z 393.48,A -85,B 0,C 180,E1 -3785.179,E2 -3785.179} C_VEL
LIN {X 0,Y 544.888,Z 400.55,A -85,B 0,C 180,E1 -3788.156,E2 -3788.156} C_VEL
LIN {X 0,Y 544.86,Z 408.256,A -85,B 0,C 180,E1 -3791.389,E2 -3791.389} C_VEL
LIN {X 0,Y 544.748,Z 415.78,A -85,B 0,C 180,E1 -3794.623,E2 -3794.623} C_VEL
LIN {X 0,Y 544.65,Z 423.377,A -85,B 0,C 180,E1 -3797.846,E2 -3797.846} C_VEL
LIN {X 0,Y 544.642,Z 423.494,A -85,B 0,C 180,E1 -3797.895,E2 -3797.895} C_VEL
LIN {X 0,Y 546.123,Z 432.591,A -85,B 0,C 180,E1 -3798.135,E2 -3798.135} C_VEL
LIN {X 0,Y 545.998,Z 442.446,A -85,B 0,C 180,E1 -3798.431,E2 -3798.431} C_VEL
LIN {X 0,Y 545.803,Z 453.426,A -85,B 0,C 180,E1 -3798.876,E2 -3798.876} C_VEL
LIN {X 0,Y 545.656,Z 463.108,A -85,B 0,C 180,E1 -3799.369,E2 -3799.369} C_VEL
LIN {X 0,Y 545.451,Z 473.339,A -85,B 0,C 180,E1 -3800.034,E2 -3800.034} C_VEL
LIN {X 0,Y 545.334,Z 481.374,A -85,B 0,C 180,E1 -3800.658,E2 -3800.658} C_VEL
LIN {X 0,Y 545.19,Z 488.918,A -85,B 0,C 180,E1 -3801.346,E2 -3801.346} C_VEL
LIN {X 0,Y 545.03,Z 496.473,A -85,B 0,C 180,E1 -3802.158,E2 -3802.158} C_VEL
LIN {X 0,Y 544.93,Z 502.827,A -85,B 0,C 180,E1 -3802.963,E2 -3802.963} C_VEL
LIN {X 0,Y 544.827,Z 509.587,A -85,B 0,C 180,E1 -3803.99,E2 -3803.99} C_VEL
LIN {X 0,Y 544.734,Z 514.033,A -85,B 0,C 180,E1 -3804.79,E2 -3804.79} C_VEL
LIN {X 0,Y 544.671,Z 519.578,A -85,B 0,C 180,E1 -3806.021,E2 -3806.021} C_VEL
LIN {X 0,Y 544.654,Z 523.145,A -85,B 0,C 180,E1 -3807.082,E2 -3807.082} C_VEL
LIN {X 0,Y 544.624,Z 524.857,A -85,B 0,C 180,E1 -3807.681,E2 -3807.681} C_VEL
LIN {X 0,Y 544.599,Z 526.9,A -85,B 0,C 180,E1 -3808.653,E2 -3808.653} C_VEL
LIN {X 0,Y 544.597,Z 528.73,A -85,B 0,C 180,E1 -3810.218,E2 -3810.218} C_VEL
LIN {X 0,Y 544.544,Z 528.911,A -85,B 0,C 180,E1 -3811.488,E2 -3811.488} C_VEL
LIN {X 0,Y 543.887,Z 528.637,A -85,B 0,C 180,E1 -3812.105,E2 -3812.105} C_VEL
LIN {X 0,Y 541.04,Z 527.574,A -85,B 0,C 180,E1 -3813.102,E2 -3813.102} C_VEL
LIN {X 0,Y 538.631,Z 526.154,A -85,B 0,C 180,E1 -3813.895,E2 -3813.895} C_VEL
LIN {X 0,Y 537.596,Z 524.734,A -85,B 0,C 180,E1 -3814.5,E2 -3814.5} C_VEL
LIN {X 0,Y 537.513,Z 524.192,A -85,B 0,C 180,E1 -3814.703,E2 -3814.703} C_VEL
LIN {X 0,Y 537.581,Z 519.934,A -85,B 0,C 180,E1 -3816.036,E2 -3816.036} C_VEL
LIN {X 0,Y 537.631,Z 515.351,A -85,B 0,C 180,E1 -3817.116,E2 -3817.116} C_VEL
LIN {X 0,Y 537.743,Z 508.701,A -85,B 0,C 180,E1 -3818.355,E2 -3818.355} C_VEL
LIN {X 0,Y 537.922,Z 500.381,A -85,B 0,C 180,E1 -3819.57,E2 -3819.57} C_VEL
LIN {X 0,Y 538.093,Z 492.358,A -85,B 0,C 180,E1 -3820.521,E2 -3820.521} C_VEL
LIN {X 0,Y 538.296,Z 482.314,A -85,B 0,C 180,E1 -3821.498,E2 -3821.498} C_VEL
LIN {X 0,Y 538.472,Z 472.186,A -85,B 0,C 180,E1 -3822.291,E2 -3822.291} C_VEL
LIN {X 0,Y 538.707,Z 460.886,A -85,B 0,C 180,E1 -3822.999,E2 -3822.999} C_VEL
LIN {X 0,Y 538.914,Z 449.233,A -85,B 0,C 180,E1 -3823.569,E2 -3823.569} C_VEL
LIN {X 0,Y 539.148,Z 436.546,A -85,B 0,C 180,E1 -3824.019,E2 -3824.019} C_VEL
LIN {X 0,Y 539.001,Z 431.973,A -85,B 0,C 180,E1 -3824.151,E2 -3824.151} C_VEL
LIN {X 0,Y 537.597,Z 423.48,A -85,B 0,C 180,E1 -3824.377,E2 -3824.377} C_VEL
LIN {X 0,Y 537.639,Z 417.048,A -85,B 0,C 180,E1 -3827.176,E2 -3827.176} C_VEL
LIN {X 0,Y 537.693,Z 410.192,A -85,B 0,C 180,E1 -3830.173,E2 -3830.173} C_VEL
LIN {X 0,Y 537.753,Z 403.417,A -85,B 0,C 180,E1 -3833.044,E2 -3833.044} C_VEL
LIN {X 0,Y 537.797,Z 397.092,A -85,B 0,C 180,E1 -3835.81,E2 -3835.81} C_VEL
LIN {X 0,Y 537.875,Z 390.856,A -85,B 0,C 180,E1 -3838.489,E2 -3838.489} C_VEL
LIN {X 0,Y 537.874,Z 384.783,A -85,B 0,C 180,E1 -3841.097,E2 -3841.097} C_VEL
LIN {X 0,Y 537.923,Z 377.134,A -85,B 0,C 180,E1 -3844.354,E2 -3844.354} C_VEL
LIN {X 0,Y 538.024,Z 373.47,A -85,B 0,C 180,E1 -3845.907,E2 -3845.907} C_VEL
LIN {X 0,Y 538.024,Z 373.467,A -85,B 0,C 180,E1 -3848.545,E2 -3848.545} C_VEL
LIN {X 0,Y 538.017,Z 373.467,A -85,B 0,C 180,E1 -3850.938,E2 -3850.938} C_VEL
LIN {X 0,Y 538.013,Z 373.469,A -85,B 0,C 180,E1 -3853.297,E2 -3853.297} C_VEL
LIN {X 0,Y 538.066,Z 373.461,A -85,B 0,C 180,E1 -3855.629,E2 -3855.629} C_VEL
LIN {X 0,Y 538.077,Z 373.46,A -85,B 0,C 180,E1 -3858.7,E2 -3858.7} C_VEL
LIN {X 0,Y 538.085,Z 373.46,A -85,B 0,C 180,E1 -3861.738,E2 -3861.738} C_VEL
LIN {X 0,Y 538.152,Z 373.454,A -85,B 0,C 180,E1 -3864.753,E2 -3864.753} C_VEL
LIN {X 0,Y 538.164,Z 373.453,A -85,B 0,C 180,E1 -3867.753,E2 -3867.753} C_VEL
LIN {X 0,Y 538.176,Z 373.49,A -85,B 0,C 180,E1 -3870.372,E2 -3870.372} C_VEL
LIN {X 0,Y 538.148,Z 377.213,A -85,B 0,C 180,E1 -3872.244,E2 -3872.244} C_VEL
LIN {X 0,Y 537.97,Z 383.245,A -85,B 0,C 180,E1 -3875.245,E2 -3875.245} C_VEL
LIN {X 0,Y 537.9,Z 387.829,A -85,B 0,C 180,E1 -3877.506,E2 -3877.506} C_VEL
LIN {X 0,Y 537.825,Z 394.081,A -85,B 0,C 180,E1 -3880.539,E2 -3880.539} C_VEL
LIN {X 0,Y 537.714,Z 400.473,A -85,B 0,C 180,E1 -3883.605,E2 -3883.605} C_VEL
LIN {X 0,Y 537.647,Z 405.367,A -85,B 0,C 180,E1 -3885.931,E2 -3885.931} C_VEL
LIN {X 0,Y 537.577,Z 410.293,A -85,B 0,C 180,E1 -3888.284,E2 -3888.284} C_VEL
LIN {X 0,Y 537.541,Z 415.36,A -85,B 0,C 180,E1 -3890.669,E2 -3890.669} C_VEL
LIN {X 0,Y 537.515,Z 419.37,A -85,B 0,C 180,E1 -3892.533,E2 -3892.533} C_VEL
LIN {X 0,Y 538.569,Z 428.903,A -85,B 0,C 180,E1 -3892.841,E2 -3892.841} C_VEL
LIN {X 0,Y 538.361,Z 439.292,A -85,B 0,C 180,E1 -3893.257,E2 -3893.257} C_VEL
LIN {X 0,Y 538.205,Z 448.776,A -85,B 0,C 180,E1 -3893.774,E2 -3893.774} C_VEL
LIN {X 0,Y 538.075,Z 457.286,A -85,B 0,C 180,E1 -3894.364,E2 -3894.364} C_VEL
LIN {X 0,Y 537.946,Z 465.991,A -85,B 0,C 180,E1 -3895.123,E2 -3895.123} C_VEL
LIN {X 0,Y 537.834,Z 471.957,A -85,B 0,C 180,E1 -3895.746,E2 -3895.746} C_VEL
LIN {X 0,Y 537.75,Z 478.574,A -85,B 0,C 180,E1 -3896.589,E2 -3896.589} C_VEL
LIN {X 0,Y 537.683,Z 483.877,A -85,B 0,C 180,E1 -3897.412,E2 -3897.412} C_VEL
LIN {X 0,Y 537.643,Z 487.458,A -85,B 0,C 180,E1 -3898.07,E2 -3898.07} C_VEL
LIN {X 0,Y 537.572,Z 491.228,A -85,B 0,C 180,E1 -3898.926,E2 -3898.926} C_VEL
LIN {X 0,Y 537.543,Z 494.174,A -85,B 0,C 180,E1 -3899.787,E2 -3899.787} C_VEL
LIN {X 0,Y 537.482,Z 496.391,A -85,B 0,C 180,E1 -3900.658,E2 -3900.658} C_VEL
LIN {X 0,Y 537.452,Z 498.26,A -85,B 0,C 180,E1 -3901.792,E2 -3901.792} C_VEL
LIN {X 0,Y 537.458,Z 498.965,A -85,B 0,C 180,E1 -3903.188,E2 -3903.188} C_VEL
LIN {X 0,Y 537.471,Z 497.937,A -85,B 0,C 180,E1 -3904.534,E2 -3904.534} C_VEL
LIN {X 0,Y 537.464,Z 497.082,A -85,B 0,C 180,E1 -3905.121,E2 -3905.121} C_VEL
LIN {X 0,Y 537.547,Z 494.982,A -85,B 0,C 180,E1 -3906.036,E2 -3906.036} C_VEL
LIN {X 0,Y 537.582,Z 491.441,A -85,B 0,C 180,E1 -3907.111,E2 -3907.111} C_VEL
LIN {X 0,Y 537.632,Z 486.905,A -85,B 0,C 180,E1 -3908.127,E2 -3908.127} C_VEL
LIN {X 0,Y 537.706,Z 481.789,A -85,B 0,C 180,E1 -3909.027,E2 -3909.027} C_VEL
LIN {X 0,Y 537.824,Z 474.334,A -85,B 0,C 180,E1 -3910.055,E2 -3910.055} C_VEL
LIN {X 0,Y 537.9,Z 467.81,A -85,B 0,C 180,E1 -3910.786,E2 -3910.786} C_VEL
LIN {X 0,Y 538.025,Z 461.308,A -85,B 0,C 180,E1 -3911.395,E2 -3911.395} C_VEL
LIN {X 0,Y 538.197,Z 452.619,A -85,B 0,C 180,E1 -3912.058,E2 -3912.058} C_VEL
LIN {X 0,Y 538.338,Z 444.187,A -85,B 0,C 180,E1 -3912.574,E2 -3912.574} C_VEL
LIN {X 0,Y 538.458,Z 436.068,A -85,B 0,C 180,E1 -3912.969,E2 -3912.969} C_VEL
LIN {X 0,Y 538.486,Z 426.695,A -85,B 0,C 180,E1 -3913.317,E2 -3913.317} C_VEL
LIN {X 0,Y 537.573,Z 419.389,A -85,B 0,C 180,E1 -3913.55,E2 -3913.55} C_VEL
LIN {X 0,Y 537.603,Z 413.848,A -85,B 0,C 180,E1 -3916.143,E2 -3916.143} C_VEL
LIN {X 0,Y 537.627,Z 407.227,A -85,B 0,C 180,E1 -3919.301,E2 -3919.301} C_VEL
LIN {X 0,Y 537.711,Z 401.444,A -85,B 0,C 180,E1 -3922.099,E2 -3922.099} C_VEL
LIN {X 0,Y 537.745,Z 395.56,A -85,B 0,C 180,E1 -3924.897,E2 -3924.897} C_VEL
LIN {X 0,Y 537.818,Z 389.998,A -85,B 0,C 180,E1 -3927.604,E2 -3927.604} C_VEL
LIN {X 0,Y 537.905,Z 384.647,A -85,B 0,C 180,E1 -3930.232,E2 -3930.232} C_VEL
LIN {X 0,Y 538.009,Z 379.442,A -85,B 0,C 180,E1 -3932.793,E2 -3932.793} C_VEL
LIN {X 0,Y 538.095,Z 374.412,A -85,B 0,C 180,E1 -3935.295,E2 -3935.295} C_VEL
LIN {X 0,Y 538.061,Z 373.465,A -85,B 0,C 180,E1 -3935.818,E2 -3935.818} C_VEL
LIN {X 0,Y 538.016,Z 373.468,A -85,B 0,C 180,E1 -3938.546,E2 -3938.546} C_VEL
LIN {X 0,Y 538.02,Z 373.47,A -85,B 0,C 180,E1 -3940.94,E2 -3940.94} C_VEL
LIN {X 0,Y 538.006,Z 373.474,A -85,B 0,C 180,E1 -3943.299,E2 -3943.299} C_VEL
LIN {X 0,Y 538.046,Z 373.466,A -85,B 0,C 180,E1 -3945.63,E2 -3945.63} C_VEL
LIN {X 0,Y 538.086,Z 373.463,A -85,B 0,C 180,E1 -3948.702,E2 -3948.702} C_VEL
LIN {X 0,Y 538.069,Z 373.461,A -85,B 0,C 180,E1 -3951.74,E2 -3951.74} C_VEL
LIN {X 0,Y 538.17,Z 373.449,A -85,B 0,C 180,E1 -3954.755,E2 -3954.755} C_VEL
LIN {X 0,Y 538.152,Z 373.453,A -85,B 0,C 180,E1 -3957.755,E2 -3957.755} C_VEL
LIN {X 0,Y 538.168,Z 373.451,A -85,B 0,C 180,E1 -3960.749,E2 -3960.749} C_VEL
LIN {X 0,Y 538.124,Z 373.455,A -85,B 0,C 180,E1 -3962.995,E2 -3962.995} C_VEL
LIN {X 0,Y 538.115,Z 373.458,A -85,B 0,C 180,E1 -3965.998,E2 -3965.998} C_VEL
LIN {X 0,Y 538.06,Z 373.462,A -85,B 0,C 180,E1 -3969.018,E2 -3969.018} C_VEL
LIN {X 0,Y 538.062,Z 373.461,A -85,B 0,C 180,E1 -3972.063,E2 -3972.063} C_VEL
LIN {X 0,Y 538.024,Z 373.469,A -85,B 0,C 180,E1 -3975.145,E2 -3975.145} C_VEL
LIN {X 0,Y 538.07,Z 373.461,A -85,B 0,C 180,E1 -3977.553,E2 -3977.553} C_VEL
LIN {X 0,Y 538.022,Z 373.47,A -85,B 0,C 180,E1 -3980.652,E2 -3980.652} C_VEL
LIN {X 0,Y 538.022,Z 373.468,A -85,B 0,C 180,E1 -3983.072,E2 -3983.072} C_VEL
LIN {X 0,Y 538.028,Z 373.467,A -85,B 0,C 180,E1 -3985.675,E2 -3985.675} C_VEL
LIN {X 0,Y 538.029,Z 373.466,A -85,B 0,C 180,E1 -3988.051,E2 -3988.051} C_VEL
LIN {X 0,Y 538.009,Z 373.468,A -85,B 0,C 180,E1 -3990.628,E2 -3990.628} C_VEL
LIN {X 0,Y 538.025,Z 373.466,A -85,B 0,C 180,E1 -3993.285,E2 -3993.285} C_VEL
LIN {X 0,Y 538.01,Z 373.468,A -85,B 0,C 180,E1 -3996.004,E2 -3996.004} C_VEL
LIN {X 0,Y 538,Z 373.47,A -85,B 0,C 180,E1 -3998.832,E2 -3998.832} C_VEL
LIN {X 0,Y 538.062,Z 373.466,A -85,B 0,C 180,E1 -4000.775,E2 -4000.775} C_VEL
LIN {X 0,Y 538.015,Z 373.468,A -85,B 0,C 180,E1 -4004.077,E2 -4004.077} C_VEL
LIN {X 0,Y 538.01,Z 373.47,A -85,B 0,C 180,E1 -4007.217,E2 -4007.217} C_VEL
LIN {X 0,Y 538.043,Z 373.468,A -85,B 0,C 180,E1 -4010.208,E2 -4010.208} C_VEL
LIN {X 0,Y 538.019,Z 373.47,A -85,B 0,C 180,E1 -4013.07,E2 -4013.07} C_VEL
LIN {X 0,Y 538.024,Z 373.469,A -85,B 0,C 180,E1 -4015.83,E2 -4015.83} C_VEL
LIN {X 0,Y 538.07,Z 373.652,A -85,B 0,C 180,E1 -4017.972,E2 -4017.972} C_VEL
LIN {X 0,Y 539.23,Z 380.351,A -85,B 0,C 180,E1 -4019.885,E2 -4019.885} C_VEL
LIN {X 0,Y 539.01,Z 390.184,A -85,B 0,C 180,E1 -4022.454,E2 -4022.454} C_VEL
LIN {X 0,Y 538.615,Z 403.016,A -85,B 0,C 180,E1 -4025.703,E2 -4025.703} C_VEL
LIN {X 0,Y 538.381,Z 413.555,A -85,B 0,C 180,E1 -4028.253,E2 -4028.253} C_VEL
LIN {X 0,Y 538.211,Z 425.217,A -85,B 0,C 180,E1 -4030.949,E2 -4030.949} C_VEL
LIN {X 0,Y 538.072,Z 437.234,A -85,B 0,C 180,E1 -4033.693,E2 -4033.693} C_VEL
LIN {X 0,Y 537.881,Z 449.138,A -85,B 0,C 180,E1 -4036.399,E2 -4036.399} C_VEL
LIN {X 0,Y 537.86,Z 450.137,A -85,B 0,C 180,E1 -4036.627,E2 -4036.627} C_VEL
LIN {X 0,Y 539.258,Z 459.595,A -85,B 0,C 180,E1 -4036.842,E2 -4036.842} C_VEL
LIN {X 0,Y 539.102,Z 471.919,A -85,B 0,C 180,E1 -4037.198,E2 -4037.198} C_VEL
LIN {X 0,Y 538.899,Z 483.54,A -85,B 0,C 180,E1 -4037.671,E2 -4037.671} C_VEL
LIN {X 0,Y 538.649,Z 495.107,A -85,B 0,C 180,E1 -4038.291,E2 -4038.291} C_VEL
LIN {X 0,Y 538.463,Z 506.768,A -85,B 0,C 180,E1 -4039.093,E2 -4039.093} C_VEL
LIN {X 0,Y 538.2,Z 517.617,A -85,B 0,C 180,E1 -4040.038,E2 -4040.038} C_VEL
LIN {X 0,Y 538.013,Z 526.429,A -85,B 0,C 180,E1 -4040.983,E2 -4040.983} C_VEL
LIN {X 0,Y 537.827,Z 535.016,A -85,B 0,C 180,E1 -4042.116,E2 -4042.116} C_VEL
LIN {X 0,Y 537.704,Z 541.879,A -85,B 0,C 180,E1 -4043.246,E2 -4043.246} C_VEL
LIN {X 0,Y 537.676,Z 547.373,A -85,B 0,C 180,E1 -4044.376,E2 -4044.376} C_VEL
LIN {X 0,Y 537.557,Z 551.683,A -85,B 0,C 180,E1 -4045.503,E2 -4045.503} C_VEL
LIN {X 0,Y 537.591,Z 553.966,A -85,B 0,C 180,E1 -4046.254,E2 -4046.254} C_VEL
LIN {X 0,Y 537.551,Z 555.814,A -85,B 0,C 180,E1 -4047.004,E2 -4047.004} C_VEL
LIN {X 0,Y 537.451,Z 558.186,A -85,B 0,C 180,E1 -4048.503,E2 -4048.503} C_VEL
LIN {X 0,Y 537.442,Z 559,A -85,B 0,C 180,E1 -4050.002,E2 -4050.002} C_VEL
LIN {X 0,Y 537.451,Z 558.181,A -85,B 0,C 180,E1 -4051.5,E2 -4051.5} C_VEL
LIN {X 0,Y 537.551,Z 555.804,A -85,B 0,C 180,E1 -4052.999,E2 -4052.999} C_VEL
LIN {X 0,Y 537.604,Z 552.89,A -85,B 0,C 180,E1 -4054.125,E2 -4054.125} C_VEL
LIN {X 0,Y 537.588,Z 548.944,A -85,B 0,C 180,E1 -4055.252,E2 -4055.252} C_VEL
LIN {X 0,Y 537.652,Z 544.089,A -85,B 0,C 180,E1 -4056.334,E2 -4056.334} C_VEL
LIN {X 0,Y 537.793,Z 537.456,A -85,B 0,C 180,E1 -4057.511,E2 -4057.511} C_VEL
LIN {X 0,Y 537.971,Z 529.466,A -85,B 0,C 180,E1 -4058.642,E2 -4058.642} C_VEL
LIN {X 0,Y 538.12,Z 521.319,A -85,B 0,C 180,E1 -4059.587,E2 -4059.587} C_VEL
LIN {X 0,Y 538.35,Z 511.382,A -85,B 0,C 180,E1 -4060.532,E2 -4060.532} C_VEL
LIN {X 0,Y 538.558,Z 501.569,A -85,B 0,C 180,E1 -4061.29,E2 -4061.29} C_VEL
LIN {X 0,Y 538.741,Z 490.592,A -85,B 0,C 180,E1 -4061.971,E2 -4061.971} C_VEL
LIN {X 0,Y 538.989,Z 478.077,A -85,B 0,C 180,E1 -4062.569,E2 -4062.569} C_VEL
LIN {X 0,Y 539.219,Z 465.044,A -85,B 0,C 180,E1 -4063.018,E2 -4063.018} C_VEL
LIN {X 0,Y 539.021,Z 457.164,A -85,B 0,C 180,E1 -4063.215,E2 -4063.215} C_VEL
LIN {X 0,Y 537.87,Z 450.069,A -85,B 0,C 180,E1 -4063.388,E2 -4063.388} C_VEL
LIN {X 0,Y 538.076,Z 437.294,A -85,B 0,C 180,E1 -4066.31,E2 -4066.31} C_VEL
LIN {X 0,Y 538.27,Z 423.727,A -85,B 0,C 180,E1 -4069.449,E2 -4069.449} C_VEL
LIN {X 0,Y 538.514,Z 410.139,A -85,B 0,C 180,E1 -4072.645,E2 -4072.645} C_VEL
LIN {X 0,Y 538.759,Z 398.397,A -85,B 0,C 180,E1 -4075.499,E2 -4075.499} C_VEL
LIN {X 0,Y 539.108,Z 386.845,A -85,B 0,C 180,E1 -4078.414,E2 -4078.414} C_VEL
LIN {X 0,Y 539.224,Z 380.289,A -85,B 0,C 180,E1 -4080.12,E2 -4080.12} C_VEL
LIN {X 0,Y 538.05,Z 373.463,A -85,B 0,C 180,E1 -4082.033,E2 -4082.033} C_VEL
LIN {X 0,Y 538.019,Z 373.47,A -85,B 0,C 180,E1 -4084.618,E2 -4084.618} C_VEL
LIN {X 0,Y 538.006,Z 373.467,A -85,B 0,C 180,E1 -4087.17,E2 -4087.17} C_VEL
LIN {X 0,Y 538.013,Z 373.471,A -85,B 0,C 180,E1 -4089.799,E2 -4089.799} C_VEL
LIN {X 0,Y 537.964,Z 373.471,A -85,B 0,C 180,E1 -4092.792,E2 -4092.792} C_VEL
LIN {X 0,Y 537.994,Z 373.472,A -85,B 0,C 180,E1 -4095.136,E2 -4095.136} C_VEL
LIN {X 0,Y 538.004,Z 373.466,A -85,B 0,C 180,E1 -4098.224,E2 -4098.224} C_VEL
LIN {X 0,Y 538.016,Z 373.465,A -85,B 0,C 180,E1 -4101.169,E2 -4101.169} C_VEL
LIN {X 0,Y 538,Z 373.47,A -85,B 0,C 180,E1 -4104.089,E2 -4104.089} C_VEL
LIN {X 0,Y 538.036,Z 373.462,A -85,B 0,C 180,E1 -4106.727,E2 -4106.727} C_VEL
LIN {X 0,Y 538.011,Z 373.47,A -85,B 0,C 180,E1 -4109.56,E2 -4109.56} C_VEL
LIN {X 0,Y 537.996,Z 373.468,A -85,B 0,C 180,E1 -4112.662,E2 -4112.662} C_VEL
LIN {X 0,Y 537.971,Z 373.475,A -85,B 0,C 180,E1 -4115.288,E2 -4115.288} C_VEL
LIN {X 0,Y 538.019,Z 373.465,A -85,B 0,C 180,E1 -4118.042,E2 -4118.042} C_VEL
LIN {X 0,Y 538.036,Z 373.464,A -85,B 0,C 180,E1 -4120.94,E2 -4120.94} C_VEL
LIN {X 0,Y 538.027,Z 373.464,A -85,B 0,C 180,E1 -4123.299,E2 -4123.299} C_VEL
LIN {X 0,Y 538.067,Z 373.464,A -85,B 0,C 180,E1 -4125.631,E2 -4125.631} C_VEL
LIN {X 0,Y 538.075,Z 373.458,A -85,B 0,C 180,E1 -4128.701,E2 -4128.701} C_VEL
LIN {X 0,Y 538.035,Z 373.464,A -85,B 0,C 180,E1 -4131.739,E2 -4131.739} C_VEL
LIN {X 0,Y 538.146,Z 373.456,A -85,B 0,C 180,E1 -4134.755,E2 -4134.755} C_VEL
LIN {X 0,Y 537.78,Z 373.618,A -85,B 0,C 180,E1 -4137.05,E2 -4137.05} C_VEL
LIN {X 0,Y 537.964,Z 381.255,A -85,B 0,C 180,E1 -4140,E2 -4140} C_VEL
LIN {X 0,Y 537.796,Z 386.947,A -85,B 0,C 180,E1 -4142.247,E2 -4142.247} C_VEL
LIN {X 0,Y 537.877,Z 394.318,A -85,B 0,C 180,E1 -4145.248,E2 -4145.248} C_VEL
LIN {X 0,Y 537.817,Z 401.534,A -85,B 0,C 180,E1 -4148.264,E2 -4148.264} C_VEL
LIN {X 0,Y 537.779,Z 409.001,A -85,B 0,C 180,E1 -4151.436,E2 -4151.436} C_VEL
LIN {X 0,Y 537.676,Z 416.585,A -85,B 0,C 180,E1 -4154.701,E2 -4154.701} C_VEL
LIN {X 0,Y 537.578,Z 423.517,A -85,B 0,C 180,E1 -4157.728,E2 -4157.728} C_VEL
LIN {X 0,Y 539.212,Z 433.316,A -85,B 0,C 180,E1 -4157.988,E2 -4157.988} C_VEL
LIN {X 0,Y 539.06,Z 442.879,A -85,B 0,C 180,E1 -4158.283,E2 -4158.283} C_VEL
LIN {X 0,Y 538.906,Z 452.686,A -85,B 0,C 180,E1 -4158.682,E2 -4158.682} C_VEL
LIN {X 0,Y 538.702,Z 463.398,A -85,B 0,C 180,E1 -4159.233,E2 -4159.233} C_VEL
LIN {X 0,Y 538.466,Z 473.37,A -85,B 0,C 180,E1 -4159.893,E2 -4159.893} C_VEL
LIN {X 0,Y 538.333,Z 481.648,A -85,B 0,C 180,E1 -4160.546,E2 -4160.546} C_VEL
LIN {X 0,Y 538.147,Z 489.202,A -85,B 0,C 180,E1 -4161.248,E2 -4161.248} C_VEL
LIN {X 0,Y 537.986,Z 496.703,A -85,B 0,C 180,E1 -4162.07,E2 -4162.07} C_VEL
LIN {X 0,Y 537.873,Z 502.947,A -85,B 0,C 180,E1 -4162.875,E2 -4162.875} C_VEL
LIN {X 0,Y 537.761,Z 509.591,A -85,B 0,C 180,E1 -4163.9,E2 -4163.9} C_VEL
LIN {X 0,Y 537.644,Z 514.117,A -85,B 0,C 180,E1 -4164.727,E2 -4164.727} C_VEL
LIN {X 0,Y 537.583,Z 519.648,A -85,B 0,C 180,E1 -4165.973,E2 -4165.973} C_VEL
LIN {X 0,Y 537.558,Z 523.766,A -85,B 0,C 180,E1 -4167.248,E2 -4167.248} C_VEL
LIN {X 0,Y 537.496,Z 525.805,A -85,B 0,C 180,E1 -4168.081,E2 -4168.081} C_VEL
LIN {X 0,Y 537.487,Z 527.404,A -85,B 0,C 180,E1 -4168.934,E2 -4168.934} C_VEL
LIN {X 0,Y 537.508,Z 528.815,A -85,B 0,C 180,E1 -4170.348,E2 -4170.348} C_VEL
LIN {X 0,Y 537.457,Z 528.787,A -85,B 0,C 180,E1 -4171.791,E2 -4171.791} C_VEL
LIN {X 0,Y 537.469,Z 527.171,A -85,B 0,C 180,E1 -4173.312,E2 -4173.312} C_VEL
LIN {X 0,Y 537.513,Z 524.192,A -85,B 0,C 180,E1 -4174.703,E2 -4174.703} C_VEL
LIN {X 0,Y 536.857,Z 522.492,A -85,B 0,C 180,E1 -4175.301,E2 -4175.301} C_VEL
LIN {X 0,Y 534.051,Z 519.235,A -85,B 0,C 180,E1 -4176.258,E2 -4176.258} C_VEL
LIN {X 0,Y 531.248,Z 515.336,A -85,B 0,C 180,E1 -4177.196,E2 -4177.196} C_VEL
LIN {X 0,Y 530.61,Z 512.566,A -85,B 0,C 180,E1 -4177.759,E2 -4177.759} C_VEL
LIN {X 0,Y 530.739,Z 505.202,A -85,B 0,C 180,E1 -4179.008,E2 -4179.008} C_VEL
LIN {X 0,Y 530.929,Z 497.053,A -85,B 0,C 180,E1 -4180.106,E2 -4180.106} C_VEL
LIN {X 0,Y 531.168,Z 487.068,A -85,B 0,C 180,E1 -4181.197,E2 -4181.197} C_VEL
LIN {X 0,Y 531.408,Z 477.242,A -85,B 0,C 180,E1 -4182.061,E2 -4182.061} C_VEL
LIN {X 0,Y 531.638,Z 465.215,A -85,B 0,C 180,E1 -4182.906,E2 -4182.906} C_VEL
LIN {X 0,Y 531.891,Z 453.803,A -85,B 0,C 180,E1 -4183.53,E2 -4183.53} C_VEL
LIN {X 0,Y 532.169,Z 440.659,A -85,B 0,C 180,E1 -4184.06,E2 -4184.06} C_VEL
LIN {X 0,Y 532.101,Z 433.003,A -85,B 0,C 180,E1 -4184.298,E2 -4184.298} C_VEL
LIN {X 0,Y 530.519,Z 423.55,A -85,B 0,C 180,E1 -4184.571,E2 -4184.571} C_VEL
LIN {X 0,Y 530.564,Z 416.912,A -85,B 0,C 180,E1 -4187.501,E2 -4187.501} C_VEL
LIN {X 0,Y 530.63,Z 410.765,A -85,B 0,C 180,E1 -4190.191,E2 -4190.191} C_VEL
LIN {X 0,Y 530.678,Z 403.262,A -85,B 0,C 180,E1 -4193.418,E2 -4193.418} C_VEL
LIN {X 0,Y 530.756,Z 396.868,A -85,B 0,C 180,E1 -4196.21,E2 -4196.21} C_VEL
LIN {X 0,Y 530.819,Z 390.665,A -85,B 0,C 180,E1 -4198.911,E2 -4198.911} C_VEL
LIN {X 0,Y 530.843,Z 383.587,A -85,B 0,C 180,E1 -4201.965,E2 -4201.965} C_VEL
LIN {X 0,Y 530.89,Z 376.616,A -85,B 0,C 180,E1 -4204.935,E2 -4204.935} C_VEL
LIN {X 0,Y 531.007,Z 374.344,A -85,B 0,C 180,E1 -4205.955,E2 -4205.955} C_VEL
LIN {X 0,Y 531,Z 374.344,A -85,B 0,C 180,E1 -4209.061,E2 -4209.061} C_VEL
LIN {X 0,Y 530.973,Z 374.344,A -85,B 0,C 180,E1 -4211.477,E2 -4211.477} C_VEL
LIN {X 0,Y 530.997,Z 374.341,A -85,B 0,C 180,E1 -4214.649,E2 -4214.649} C_VEL
LIN {X 0,Y 531.031,Z 374.337,A -85,B 0,C 180,E1 -4217.773,E2 -4217.773} C_VEL
LIN {X 0,Y 531.02,Z 374.338,A -85,B 0,C 180,E1 -4220.86,E2 -4220.86} C_VEL
LIN {X 0,Y 531.017,Z 374.343,A -85,B 0,C 180,E1 -4223.157,E2 -4223.157} C_VEL
LIN {X 0,Y 531.112,Z 374.332,A -85,B 0,C 180,E1 -4224.684,E2 -4224.684} C_VEL
LIN {X 0,Y 531.135,Z 374.328,A -85,B 0,C 180,E1 -4227.723,E2 -4227.723} C_VEL
LIN {X 0,Y 531.148,Z 374.459,A -85,B 0,C 180,E1 -4230.377,E2 -4230.377} C_VEL
LIN {X 0,Y 531.114,Z 378.188,A -85,B 0,C 180,E1 -4232.273,E2 -4232.273} C_VEL
LIN {X 0,Y 530.923,Z 384.248,A -85,B 0,C 180,E1 -4235.315,E2 -4235.315} C_VEL
LIN {X 0,Y 530.826,Z 390.426,A -85,B 0,C 180,E1 -4238.372,E2 -4238.372} C_VEL
LIN {X 0,Y 530.765,Z 396.832,A -85,B 0,C 180,E1 -4241.522,E2 -4241.522} C_VEL
LIN {X 0,Y 530.658,Z 403.657,A -85,B 0,C 180,E1 -4244.805,E2 -4244.805} C_VEL
LIN {X 0,Y 530.532,Z 409.753,A -85,B 0,C 180,E1 -4247.737,E2 -4247.737} C_VEL
LIN {X 0,Y 530.474,Z 414.791,A -85,B 0,C 180,E1 -4250.147,E2 -4250.147} C_VEL
LIN {X 0,Y 530.448,Z 419.543,A -85,B 0,C 180,E1 -4252.376,E2 -4252.376} C_VEL
LIN {X 0,Y 531.636,Z 429.253,A -85,B 0,C 180,E1 -4252.694,E2 -4252.694} C_VEL
LIN {X 0,Y 531.377,Z 440.622,A -85,B 0,C 180,E1 -4253.168,E2 -4253.168} C_VEL
LIN {X 0,Y 531.199,Z 449.599,A -85,B 0,C 180,E1 -4253.677,E2 -4253.677} C_VEL
LIN {X 0,Y 531.057,Z 458.521,A -85,B 0,C 180,E1 -4254.322,E2 -4254.322} C_VEL
LIN {X 0,Y 530.945,Z 465.652,A -85,B 0,C 180,E1 -4254.953,E2 -4254.953} C_VEL
LIN {X 0,Y 530.804,Z 472.087,A -85,B 0,C 180,E1 -4255.636,E2 -4255.636} C_VEL
LIN {X 0,Y 530.683,Z 479.048,A -85,B 0,C 180,E1 -4256.546,E2 -4256.546} C_VEL
LIN {X 0,Y 530.578,Z 484.587,A -85,B 0,C 180,E1 -4257.443,E2 -4257.443} C_VEL
LIN {X 0,Y 530.553,Z 487.785,A -85,B 0,C 180,E1 -4258.048,E2 -4258.048} C_VEL
LIN {X 0,Y 530.492,Z 491.91,A -85,B 0,C 180,E1 -4259.03,E2 -4259.03} C_VEL
LIN {X 0,Y 530.45,Z 495.513,A -85,B 0,C 180,E1 -4260.227,E2 -4260.227} C_VEL
LIN {X 0,Y 530.378,Z 497.387,A -85,B 0,C 180,E1 -4261.114,E2 -4261.114} C_VEL
LIN {X 0,Y 530.363,Z 498.547,A -85,B 0,C 180,E1 -4262.006,E2 -4262.006} C_VEL
LIN {X 0,Y 530.346,Z 498.976,A -85,B 0,C 180,E1 -4262.907,E2 -4262.907} C_VEL
LIN {X 0,Y 530.372,Z 498.695,A -85,B 0,C 180,E1 -4263.814,E2 -4263.814} C_VEL
LIN {X 0,Y 530.363,Z 497.68,A -85,B 0,C 180,E1 -4264.757,E2 -4264.757} C_VEL
LIN {X 0,Y 530.47,Z 495.005,A -85,B 0,C 180,E1 -4266.083,E2 -4266.083} C_VEL
LIN {X 0,Y 530.504,Z 490.722,A -85,B 0,C 180,E1 -4267.358,E2 -4267.358} C_VEL
LIN {X 0,Y 530.564,Z 486.68,A -85,B 0,C 180,E1 -4268.259,E2 -4268.259} C_VEL
LIN {X 0,Y 530.649,Z 481.099,A -85,B 0,C 180,E1 -4269.236,E2 -4269.236} C_VEL
LIN {X 0,Y 530.789,Z 474.937,A -85,B 0,C 180,E1 -4270.103,E2 -4270.103} C_VEL
LIN {X 0,Y 530.876,Z 468.186,A -85,B 0,C 180,E1 -4270.881,E2 -4270.881} C_VEL
LIN {X 0,Y 531.028,Z 461.085,A -85,B 0,C 180,E1 -4271.555,E2 -4271.555} C_VEL
LIN {X 0,Y 531.213,Z 452.838,A -85,B 0,C 180,E1 -4272.194,E2 -4272.194} C_VEL
LIN {X 0,Y 531.37,Z 444.08,A -85,B 0,C 180,E1 -4272.736,E2 -4272.736} C_VEL
LIN {X 0,Y 531.506,Z 434.974,A -85,B 0,C 180,E1 -4273.175,E2 -4273.175} C_VEL
LIN {X 0,Y 531.406,Z 426.551,A -85,B 0,C 180,E1 -4273.487,E2 -4273.487} C_VEL
LIN {X 0,Y 530.472,Z 419.574,A -85,B 0,C 180,E1 -4273.706,E2 -4273.706} C_VEL
LIN {X 0,Y 530.527,Z 413.138,A -85,B 0,C 180,E1 -4276.765,E2 -4276.765} C_VEL
LIN {X 0,Y 530.558,Z 407.434,A -85,B 0,C 180,E1 -4279.528,E2 -4279.528} C_VEL
LIN {X 0,Y 530.638,Z 401.394,A -85,B 0,C 180,E1 -4282.465,E2 -4282.465} C_VEL
LIN {X 0,Y 530.713,Z 395.546,A -85,B 0,C 180,E1 -4285.29,E2 -4285.29} C_VEL
LIN {X 0,Y 530.8,Z 389.974,A -85,B 0,C 180,E1 -4288.021,E2 -4288.021} C_VEL
LIN {X 0,Y 530.889,Z 384.203,A -85,B 0,C 180,E1 -4290.888,E2 -4290.888} C_VEL
LIN {X 0,Y 530.981,Z 379.48,A -85,B 0,C 180,E1 -4293.255,E2 -4293.255} C_VEL
LIN {X 0,Y 531.021,Z 374.342,A -85,B 0,C 180,E1 -4295.839,E2 -4295.839} C_VEL
LIN {X 0,Y 530.985,Z 374.347,A -85,B 0,C 180,E1 -4299.062,E2 -4299.062} C_VEL
LIN {X 0,Y 530.992,Z 374.345,A -85,B 0,C 180,E1 -4302.277,E2 -4302.277} C_VEL
LIN {X 0,Y 531.019,Z 374.34,A -85,B 0,C 180,E1 -4305.436,E2 -4305.436} C_VEL
LIN {X 0,Y 531.037,Z 374.34,A -85,B 0,C 180,E1 -4308.55,E2 -4308.55} C_VEL
LIN {X 0,Y 531.038,Z 374.338,A -85,B 0,C 180,E1 -4311.629,E2 -4311.629} C_VEL
LIN {X 0,Y 531.125,Z 374.326,A -85,B 0,C 180,E1 -4314.686,E2 -4314.686} C_VEL
LIN {X 0,Y 531.124,Z 374.328,A -85,B 0,C 180,E1 -4317.725,E2 -4317.725} C_VEL
LIN {X 0,Y 531.137,Z 374.326,A -85,B 0,C 180,E1 -4320.758,E2 -4320.758} C_VEL
LIN {X 0,Y 531.09,Z 374.332,A -85,B 0,C 180,E1 -4323.034,E2 -4323.034} C_VEL
LIN {X 0,Y 531.072,Z 374.334,A -85,B 0,C 180,E1 -4326.077,E2 -4326.077} C_VEL
LIN {X 0,Y 531.019,Z 374.338,A -85,B 0,C 180,E1 -4329.139,E2 -4329.139} C_VEL
LIN {X 0,Y 531.044,Z 374.336,A -85,B 0,C 180,E1 -4331.682,E2 -4331.682} C_VEL
LIN {X 0,Y 531.007,Z 374.341,A -85,B 0,C 180,E1 -4334.957,E2 -4334.957} C_VEL
LIN {X 0,Y 531.006,Z 374.342,A -85,B 0,C 180,E1 -4337.723,E2 -4337.723} C_VEL
LIN {X 0,Y 530.986,Z 374.343,A -85,B 0,C 180,E1 -4340.939,E2 -4340.939} C_VEL
LIN {X 0,Y 530.986,Z 374.342,A -85,B 0,C 180,E1 -4344.046,E2 -4344.046} C_VEL
LIN {X 0,Y 530.992,Z 374.341,A -85,B 0,C 180,E1 -4346.745,E2 -4346.745} C_VEL
LIN {X 0,Y 530.98,Z 374.343,A -85,B 0,C 180,E1 -4349.323,E2 -4349.323} C_VEL
LIN {X 0,Y 530.961,Z 374.345,A -85,B 0,C 180,E1 -4352.105,E2 -4352.105} C_VEL
LIN {X 0,Y 530.974,Z 374.345,A -85,B 0,C 180,E1 -4354.857,E2 -4354.857} C_VEL
LIN {X 0,Y 530.949,Z 374.348,A -85,B 0,C 180,E1 -4357.509,E2 -4357.509} C_VEL
LIN {X 0,Y 530.992,Z 374.344,A -85,B 0,C 180,E1 -4360.432,E2 -4360.432} C_VEL
LIN {X 0,Y 530.954,Z 374.35,A -85,B 0,C 180,E1 -4363.496,E2 -4363.496} C_VEL
LIN {X 0,Y 530.952,Z 374.348,A -85,B 0,C 180,E1 -4366.508,E2 -4366.508} C_VEL
LIN {X 0,Y 530.996,Z 374.343,A -85,B 0,C 180,E1 -4369.572,E2 -4369.572} C_VEL
LIN {X 0,Y 530.958,Z 374.35,A -85,B 0,C 180,E1 -4372.579,E2 -4372.579} C_VEL
LIN {X 0,Y 530.995,Z 374.346,A -85,B 0,C 180,E1 -4375.314,E2 -4375.314} C_VEL
LIN {X 0,Y 531.004,Z 374.503,A -85,B 0,C 180,E1 -4377.709,E2 -4377.709} C_VEL
LIN {X 0,Y 532.168,Z 380.724,A -85,B 0,C 180,E1 -4379.534,E2 -4379.534} C_VEL
LIN {X 0,Y 532.211,Z 385.203,A -85,B 0,C 180,E1 -4380.754,E2 -4380.754} C_VEL
LIN {X 0,Y 531.894,Z 394.969,A -85,B 0,C 180,E1 -4383.307,E2 -4383.307} C_VEL
LIN {X 0,Y 531.57,Z 406.398,A -85,B 0,C 180,E1 -4386.221,E2 -4386.221} C_VEL
LIN {X 0,Y 531.291,Z 416.371,A -85,B 0,C 180,E1 -4388.67,E2 -4388.67} C_VEL
LIN {X 0,Y 531.119,Z 428.421,A -85,B 0,C 180,E1 -4391.486,E2 -4391.486} C_VEL
LIN {X 0,Y 530.968,Z 440.43,A -85,B 0,C 180,E1 -4394.258,E2 -4394.258} C_VEL
LIN {X 0,Y 530.814,Z 450.05,A -85,B 0,C 180,E1 -4396.459,E2 -4396.459} C_VEL
LIN {X 0,Y 532.341,Z 460.247,A -85,B 0,C 180,E1 -4396.693,E2 -4396.693} C_VEL
LIN {X 0,Y 532.161,Z 473.024,A -85,B 0,C 180,E1 -4397.076,E2 -4397.076} C_VEL
LIN {X 0,Y 531.915,Z 485.444,A -85,B 0,C 180,E1 -4397.604,E2 -4397.604} C_VEL
LIN {X 0,Y 531.646,Z 497.273,A -85,B 0,C 180,E1 -4398.27,E2 -4398.27} C_VEL
LIN {X 0,Y 531.408,Z 509.114,A -85,B 0,C 180,E1 -4399.139,E2 -4399.139} C_VEL
LIN {X 0,Y 531.113,Z 519.559,A -85,B 0,C 180,E1 -4400.096,E2 -4400.096} C_VEL
LIN {X 0,Y 530.929,Z 528.007,A -85,B 0,C 180,E1 -4401.054,E2 -4401.054} C_VEL
LIN {X 0,Y 530.756,Z 536.247,A -85,B 0,C 180,E1 -4402.201,E2 -4402.201} C_VEL
LIN {X 0,Y 530.594,Z 543.29,A -85,B 0,C 180,E1 -4403.423,E2 -4403.423} C_VEL
LIN {X 0,Y 530.524,Z 548.955,A -85,B 0,C 180,E1 -4404.681,E2 -4404.681} C_VEL
LIN {X 0,Y 530.522,Z 552.9,A -85,B 0,C 180,E1 -4405.824,E2 -4405.824} C_VEL
LIN {X 0,Y 530.457,Z 555.814,A -85,B 0,C 180,E1 -4406.964,E2 -4406.964} C_VEL
LIN {X 0,Y 530.411,Z 557.199,A -85,B 0,C 180,E1 -4407.724,E2 -4407.724} C_VEL
LIN {X 0,Y 530.344,Z 558.787,A -85,B 0,C 180,E1 -4409.242,E2 -4409.242} C_VEL
LIN {X 0,Y 530.342,Z 559,A -85,B 0,C 180,E1 -4410.002,E2 -4410.002} C_VEL
LIN {X 0,Y 530.361,Z 558.18,A -85,B 0,C 180,E1 -4411.52,E2 -4411.52} C_VEL
LIN {X 0,Y 530.412,Z 557.191,A -85,B 0,C 180,E1 -4412.28,E2 -4412.28} C_VEL
LIN {X 0,Y 530.457,Z 555.803,A -85,B 0,C 180,E1 -4413.039,E2 -4413.039} C_VEL
LIN {X 0,Y 530.523,Z 552.89,A -85,B 0,C 180,E1 -4414.18,E2 -4414.18} C_VEL
LIN {X 0,Y 530.525,Z 548.944,A -85,B 0,C 180,E1 -4415.322,E2 -4415.322} C_VEL
LIN {X 0,Y 530.601,Z 543.256,A -85,B 0,C 180,E1 -4416.583,E2 -4416.583} C_VEL
LIN {X 0,Y 530.76,Z 536.225,A -85,B 0,C 180,E1 -4417.802,E2 -4417.802} C_VEL
